(* IEC 61131-3 sources: beebread/doc (part 8) *)

		ELSIF X.STATE = BYTE#2 THEN (* read data *)
			index2 := index + 1; (* PCWORX Workaround *)
			IF X.R_BUF.BUFFER[index] <> ID OR X.R_BUF.BUFFER[index2] <> BYTE#13 THEN (* TYPE DWORD8 *)
				X.ERROR_ID := ID;
			ELSE
				index := index + 2;
				FOR i2 := 1 TO 8 DO;
					ra[i2] := DWORD#0;
					FOR i := 1 TO 4 DO;
						ra[i2] := ra[i2] OR BYTE_TO_DWORD(X.R_BUF.BUFFER[index]);
						ra[i2] := ROR(ra[i2],8);
						index := index + 1;
					END_FOR;
				END_FOR;
				OUT1 := ra[1];
				OUT2 := ra[2];
				OUT3 := ra[3];
				OUT4 := ra[4];
				OUT5 := ra[5];
				OUT6 := ra[6];
				OUT7 := ra[7];
				OUT8 := ra[8];
			END_IF;
		END_IF;
		X.index := index;
	END_IF;
END_IF;
END_FUNCTION_BLOCK

// Commented out for beedance: it uses REAL_TO_DW, which is commented out.
// FUNCTION_BLOCK NET_VAR_REAL8
// VAR_IN_OUT
// 	X : NET_VAR_DATA;
// END_VAR
// VAR_INPUT
// 	IN1 : REAL;
// 	IN2 : REAL;
// 	IN3 : REAL;
// 	IN4 : REAL;
// 	IN5 : REAL;
// 	IN6 : REAL;
// 	IN7 : REAL;
// 	IN8 : REAL;
// END_VAR
// VAR_OUTPUT
// 	OUT1 : REAL;
// 	OUT2 : REAL;
// 	OUT3 : REAL;
// 	OUT4 : REAL;
// 	OUT5 : REAL;
// 	OUT6 : REAL;
// 	OUT7 : REAL;
// 	OUT8 : REAL;
// 	ID : BYTE;
// END_VAR
// VAR
// 	init : BOOL;
// 	i : INT;
// 	i2 : INT;
// 	index : INT;
// 	index2 : INT;
// 	r_dw : DWORD;
// 	ra : ARRAY[1..8] OF REAL;
// END_VAR
//
// IF NOT init THEN
// 	init := TRUE;
// 	X.ID_MAX := X.ID_MAX + USINT#1;
// 	ID := USINT_TO_BYTE(X.ID_MAX);
// END_IF;
//
// IF X.STATE > BYTE#0 AND X.ERROR_ID = BYTE#0 THEN
// 	index := X.index; (* PCWORX Workaround *)
// 	IF INT_TO_UINT(index + 34) > X.BUF_SIZE THEN (* ID (1) + TYPE (1) + 8 x REAL (4) *)
// 		X.ERROR_ID := ID;
// 	ELSE
// 		IF X.STATE = BYTE#1 THEN (* write data *)
// 			ra[1] := IN1;
// 			ra[2] := IN2;
// 			ra[3] := IN3;
// 			ra[4] := IN4;
// 			ra[5] := IN5;
// 			ra[6] := IN6;
// 			ra[7] := IN7;
// 			ra[8] := IN8;
// 			X.S_BUF.BUFFER[index] := ID; (* ID *)
// 			index := index + 1;
// 			X.S_BUF.BUFFER[index] := BYTE#15; (* TYPE REAL8 *)
// 			index := index + 1;
// 			FOR i2 := 1 TO 8 DO;
// 				r_dw := REAL_TO_DW(X:=ra[i2]);
// 				FOR i := 1 TO 4 DO;
// 					X.S_BUF.BUFFER[index] := DWORD_TO_BYTE(r_dw);
// 					r_dw := ROR(r_dw,8);
// 					index := index + 1;
// 				END_FOR;
// 			END_FOR;
//
// 		ELSIF X.STATE = BYTE#2 THEN (* read data *)
// 			index2 := index + 1; (* PCWORX Workaround *)
// 			IF X.R_BUF.BUFFER[index] <> ID OR X.R_BUF.BUFFER[index2] <> BYTE#15 THEN (* TYPE REAL8 *)
// 				X.ERROR_ID := ID;
// 			ELSE
// 				index := index + 2;
// 				FOR i2 := 1 TO 8 DO;
// 					r_dw := DWORD#0;
// 					FOR i := 1 TO 4 DO;
// 						r_dw := r_dw OR BYTE_TO_DWORD(X.R_BUF.BUFFER[index]);
// 						r_dw := ROR(r_dw,8);
// 						index := index + 1;
// 					END_FOR;
// 					ra[i2] := DW_TO_REAL(X:=r_dw);
// 				END_FOR;
// 				OUT1 := ra[1];
// 				OUT2 := ra[2];
// 				OUT3 := ra[3];
// 				OUT4 := ra[4];
// 				OUT5 := ra[5];
// 				OUT6 := ra[6];
// 				OUT7 := ra[7];
// 				OUT8 := ra[8];
// 			END_IF;
// 		END_IF;
// 		X.index := index;
// 	END_IF;
// END_IF;
// END_FUNCTION_BLOCK

// Commented out for beedance: it uses _STRING_TO_BUFFER, which is commented out.
// FUNCTION_BLOCK NET_VAR_STRING
// VAR_IN_OUT
// 	IN : STRING(STRING_LENGTH);
// 	OUT : STRING(STRING_LENGTH);
// 	X : NET_VAR_DATA;
// END_VAR
// VAR_OUTPUT
// 	ID : BYTE;
// END_VAR
// VAR
// 	init : BOOL;
// 	len_str : INT;
// 	index : INT;
// 	index2 : INT;
// END_VAR
//
// IF NOT init THEN
// 	init := TRUE;
// 	X.ID_MAX := X.ID_MAX + USINT#1;
// 	ID := USINT_TO_BYTE(X.ID_MAX);
// END_IF;
//
// IF X.STATE > BYTE#0 AND X.ERROR_ID = BYTE#0 THEN
// 	index := X.index; (* PCWORX Workaround *)
// 	IF X.STATE = BYTE#1 THEN (* write data *)
// 		len_str := LEN(IN);
// 		IF INT_TO_UINT(index + 3 + len_str) > X.BUF_SIZE THEN
// 			X.ERROR_ID := ID;
// 		ELSE
// 			X.S_BUF.BUFFER[index] := ID; (* ID *)
// 			index := index + 1;
// 			X.S_BUF.BUFFER[index] := BYTE#6; (* TYPE REAL *)
// 			index := index + 1;
// 			X.S_BUF.BUFFER[index] := INT_TO_BYTE(len_str); (* number of bytes *)
// 			index := index + 1;
// 			_STRING_TO_BUFFER(STR:=IN,POS:=index,PT:=REF(X.S_BUF.BUFFER),SIZE:=X.BUF_SIZE);
// 			index := index + len_str;
// 		END_IF;
// 	ELSIF X.STATE = BYTE#2 THEN (* read data *)
// 		index2 := index + 1; (* PCWORX Workaround *)
// 		IF X.R_BUF.BUFFER[index] <> ID OR X.R_BUF.BUFFER[index2] <> BYTE#6 THEN
// 			X.ERROR_ID := ID;
// 		ELSE
// 			index := index + 2;
// 			len_str := BYTE_TO_INT(X.R_BUF.BUFFER[index]);
// 			index2 := index + 1;
// 			index := index2 + len_str;
// 			IF len_STR > 0 THEN
// 				OUT := BUFFER_TO_STRING(PT:=REF(X.R_BUF.BUFFER),SIZE:=X.BUF_SIZE,START:=INT_TO_UINT(index2),STOP:=INT_TO_UINT(index - 1));
// 			ELSE
// 				OUT := '';
// 			END_IF;
// 		END_IF;
// 	END_IF;
// 	X.index := index;
// END_IF;
// END_FUNCTION_BLOCK

// Commented out for beedance: it uses REAL_TO_DW, which is commented out.
// FUNCTION_BLOCK NET_VAR_X8
// VAR_IN_OUT
// 	X : NET_VAR_DATA;
// END_VAR
// VAR_INPUT
// 	IN_REAL1 : REAL;
// 	IN_REAL2 : REAL;
// 	IN_DINT1 : DINT;
// 	IN_DINT2 : DINT;
// 	IN_UDINT1 : UDINT;
// 	IN_UDINT2 : UDINT;
// 	IN_DWORD1 : DWORD;
// 	IN_DWORD2 : DWORD;
// END_VAR
// VAR_OUTPUT
// 	OUT_REAL1 : REAL;
// 	OUT_REAL2: REAL;
// 	OUT_DINT1 : DINT;
// 	OUT_DINT2 : DINT;
// 	OUT_UDINT1 : UDINT;
// 	OUT_UDINT2 : UDINT;
// 	OUT_DWORD1 : DWORD;
// 	OUT_DWORD2 : DWORD;
// 	ID : BYTE;
// END_VAR
// VAR
// 	init : BOOL;
// 	i : INT;
// 	i2 : INT;
// 	index : INT;
// 	index2 : INT;
// 	ra : ARRAY[1..8] OF DWORD;
// END_VAR
//
// IF NOT init THEN
// 	init := TRUE;
// 	X.ID_MAX := X.ID_MAX + USINT#1;
// 	ID := USINT_TO_BYTE(X.ID_MAX);
// END_IF;
//
// IF X.STATE > BYTE#0 AND X.ERROR_ID = BYTE#0 THEN
// 	index := X.index; (* PCWORX Workaround *)
// 	IF INT_TO_UINT(index + 34) > X.BUF_SIZE THEN  (* ID (1) + TYPE (1) + 8 x DWORD (4) *)
// 		X.ERROR_ID := ID;
// 	ELSE
// 		IF X.STATE = BYTE#1 THEN (* write data *)
// 			ra[1] := REAL_TO_DW(X:=IN_REAL1);
// 			ra[2] := REAL_TO_DW(X:=IN_REAL2);
// 			ra[3] := DINT_TO_DWORD(IN_DINT1);
// 			ra[4] := DINT_TO_DWORD(IN_DINT2);
// 			ra[5] := UDINT_TO_DWORD(IN_UDINT1);
// 			ra[6] := UDINT_TO_DWORD(IN_UDINT2);
// 			ra[7] := IN_DWORD1;
// 			ra[8] := IN_DWORD2;
// 			X.S_BUF.BUFFER[index] := ID; (* ID *)
// 			index := index + 1;
// 			X.S_BUF.BUFFER[index] := BYTE#21; (* TYPE X8 *)
// 			index := index + 1;
// 			FOR i2 := 1 TO 8 DO;
// 				FOR i := 1 TO 4 DO;
// 					X.S_BUF.BUFFER[index] := DWORD_TO_BYTE(ra[i2]);
// 					ra[i2] := ROR(ra[i2],8);
// 					index := index + 1;
// 				END_FOR;
// 			END_FOR;
//
// 		ELSIF X.STATE = BYTE#2 THEN (* read data *)
// 			index2 := index + 1; (* PCWORX Workaround *)
// 			IF X.R_BUF.BUFFER[index] <> ID OR X.R_BUF.BUFFER[index2] <> BYTE#21 THEN (* TYPE X8 *)
// 				X.ERROR_ID := ID;
// 			ELSE
// 				index := index + 2;
// 				FOR i2 := 1 TO 8 DO;
// 					ra[i2] := DWORD#0;
// 					FOR i := 1 TO 4 DO;
// 						ra[i2] := ra[i2] OR BYTE_TO_DWORD(X.R_BUF.BUFFER[index]);
// 						ra[i2] := ROR(ra[i2],8);
// 						index := index + 1;
// 					END_FOR;
// 				END_FOR;
// 				OUT_REAL1 := DW_TO_REAL(X:=ra[1]);
// 				OUT_REAL2 := DW_TO_REAL(X:=ra[2]);
// 				OUT_DINT1 := DWORD_TO_DINT(ra[3]);
// 				OUT_DINT2 := DWORD_TO_DINT(ra[4]);
// 				OUT_UDINT1 := DWORD_TO_UDINT(ra[5]);
// 				OUT_UDINT2 := DWORD_TO_UDINT(ra[6]);
// 				OUT_DWORD1 := ra[7];
// 				OUT_DWORD2 := ra[8];
// 			END_IF;
// 		END_IF;
// 		X.index := index;
// 	END_IF;
// END_IF;
// END_FUNCTION_BLOCK

FUNCTION NETWORK_VERSION : DWORD
VAR_INPUT
	IN : BOOL;
END_VAR

IF in THEN
	NETWORK_VERSION := DATE_TO_DWORD(D#2016-07-01);
ELSE
	NETWORK_VERSION := 135;
END_IF;
END_FUNCTION

// Commented out for beedance: it uses CODE, which is commented out.
// FUNCTION_BLOCK PRINT_SF
// VAR_IN_OUT
// 	PRINTF_DATA : PRINTF_DATA;
// 	STR : STRING(LOG_SIZE);
// END_VAR
// VAR
// 	pos : INT;
// 	c : INT;
// 	src : STRING(1) := '~';
// 	run : BOOL;
// END_VAR
//
// IF LEN(STR) > 0 THEN
// 	run := TRUE;
//
// 	WHILE (run) DO
// 		pos := FIND(STR,src);
// 		PRINTF_DATA[10] := '';
//
// 		IF pos = 0 THEN
// 			run:= FALSE;
// 		ELSE
// 			c := CODE(STR:=STR,POS:=pos + 1);
// 			IF ISC_NUM(INT_TO_BYTE(c)) THEN
// 				c := c - 48; (* necessary because only one var is allowed inside an index expression *)
// 				PRINTF_DATA[10] := PRINTF_DATA[c]; (* command 1-9 gives parameter index 1-9 *)
// 				(* replace parameter with text *)
// 			END_IF;
// 			IF LEN(PRINTF_DATA[10]) + LEN(STR) > LOG_SIZE THEN
// 				PRINTF_DATA[10] := '..';
// 			END_IF;
// 			(* pcworx: output and input string must be different *)
// 			PRINTF_DATA[11] := STR;
// 			STR := REPLACE(PRINTF_DATA[11],PRINTF_DATA[10],2,pos);
// 		END_IF;
// 	END_WHILE;
// END_IF;
// END_FUNCTION_BLOCK

// Commented out for beedance: it uses CODE, which is commented out.
// FUNCTION_BLOCK RC4_CRYPT_STREAM
// VAR_IN_OUT
// 	MODE : INT;
// 	KEY : STRING(40);
// 	BUF : ARRAY [0..63] OF BYTE;
// 	SIZE : UDINT;
// END_VAR
//
// VAR_OUTPUT
// 	POS : UDINT;
// END_VAR
//
// VAR
// 	sbox : ARRAY [0..255] OF BYTE;
// 	skey : ARRAY [0..255] OF BYTE;
// 	a : INT;
// 	b : INT;
// 	c : INT;
// 	d : USINT;
// 	e : USINT;
// 	end : UDINT;
// 	v : BYTE;
// END_VAR
//
// CASE MODE OF
//
// 1:	(* initialization *)
// 	b := LEN(KEY) - 1;
// 	IF b < 0 OR SIZE < 1 THEN
// 		MODE := 3;
// 		RETURN;
// 	END_IF;
//
// 	FOR a := 0 TO b DO
// 		skey[a] := CODE(KEY, a + 1);
// 		sbox[a] := INT_TO_BYTE(a);
// 	END_FOR;
//
// 	c := 0;
// 	FOR a := b + 1 TO 255 DO
// 		skey[a] := skey[c];
// 		sbox[a] := INT_TO_BYTE(a);
// 		c := c + 1;
// 		IF c > b THEN c := 0; END_IF;
// 	END_FOR;
//
// 	d := 0;
// 	FOR a := 0 TO 255 DO
// 		d := d + sbox[a] + skey[a];
// 		v := sbox[a];
// 		sbox[a] := sbox[d];
// 		sbox[d] := v;
// 	END_FOR;
//
// 	POS := 0;
// 	end := SIZE;
// 	SIZE := MIN(64,end);
// 	d := 0;
// 	e := 0;
// 	MODE := 2;
//
// 2:	(* encrypt/decrypt data *)
//
// 	b := UDINT_TO_INT(SIZE) - 1;
// 	FOR a := 0 TO b DO
// 		d := d + 1;
// 		e := e + sbox[d];
// 		v := sbox[d];
// 		sbox[d] := sbox[e];
// 		sbox[e] := v;
// 		v := sbox[d] + sbox[e];
// 		BUF[a] :=BUF[a] XOR sbox[v];
// 	END_FOR;
//
// 	POS := POS + SIZE;
// 	SIZE := MIN(64,end - POS);
//
// 	IF SIZE = 0 THEN
// 		MODE := 3;
// 	END_IF;
// END_CASE;
// END_FUNCTION_BLOCK

// Commented out for beedance: it uses BUFFER_SEARCH, which is commented out.
// FUNCTION_BLOCK READ_HTTP
// VAR_INPUT
// 	SIZE : UINT;
// 	POS : INT;
// 	SRC : STRING;
// END_VAR
// VAR_IN_OUT
// 	PT : NW_BUF_LONG;
// END_VAR
// VAR_OUTPUT
// 	READ_HTTP : STRING(STRING_LENGTH);
// END_VAR
// VAR
// 	index : INT;
// 	s1 : INT;
// 	e1 : INT;
// 	stop : INT;
// END_VAR
//
// stop := UINT_TO_INT(SIZE) - 1;
//
// IF LEN(SRC) = 0 THEN
// 	(* if there is no search term, evaluate the HTTP STATUS *)
// 	SRC := 'HTTP/'; (* new search term *)
// ELSE
// 	(* append the searched parameter text *)
// 	SRC := CONCAT(SRC,': ');
// END_IF;
//
// s1 := BUFFER_SEARCH(pt:=REF(PT),SIZE:=SIZE,STR:=SRC,POS:=POS,IGN:=TRUE);
//
// IF s1 >= 0 THEN (* Text found *)
// 	e1 := s1;
//
// 	(* search start of line *)
// 	index := s1 - 1;
// 	WHILE (index > 0) DO
// 		IF pt[index] < BYTE#32 THEN EXIT; END_IF;
// 		s1 := s1 - 1;
// 		index := index - 1;
// 	END_WHILE;
//
// 	(* search end of line *)
// 	index := e1 + 1;
// 	WHILE (index <= stop) DO
// 		IF pt[index] < BYTE#32 THEN EXIT; END_IF;
// 		e1 := e1 + 1;
// 		index := index + 1;
// 	END_WHILE;
//
// 	s1 := s1 + LEN(SRC); (* do not copy 'search term: ' *)
//
// 	(* copy string *)
// 	READ_HTTP := BUFFER_TO_STRING(PT:=REF(PT),SIZE:=SIZE,START:=s1,STOP:=e1);
// ELSE
// 	READ_HTTP := '';
// END_IF;
// END_FUNCTION_BLOCK

// Commented out for beedance: it uses _STRING_TO_BUFFER, which is commented out.
// FUNCTION_BLOCK SHA1_STR
// VAR_INPUT
// 	RUN: BOOL;
// END_VAR
// VAR_OUTPUT
// 	DONE: BOOL;
// END_VAR
// VAR_IN_OUT
// 	STR: STRING(STRING_LENGTH);
// 	SHA1 : ARRAY [0..19] OF BYTE;
// END_VAR
//
// VAR
// 	run_last: BOOL;
// 	SHA1_STREAM : SHA1_STREAM;
// 	buf : ARRAY [0..63] OF BYTE;
// 	mode : INT;
// 	size : UDINT;
// 	pos : UDINT;
// END_VAR
//
// CASE mode OF
// 0:	(* wait for start *)
// 	IF RUN AND NOT run_last THEN
// 		DONE := FALSE;
// 		mode := 1; (* initialization *)
// 		size := LEN(STR);
// 	END_IF;
//
// 2:	(* Data copy and Calc *)
// 	IF size > 0 THEN
// 		_STRING_TO_BUFFER(STR:=MID(STR, UDINT_TO_INT(SIZE), UDINT_TO_INT(POS) + 1), POS:=0, PT:=REF(buf), SIZE:=SIZEOF(buf));
// 	END_IF;
//
// 3:	DONE := TRUE;
// 	mode := 0; (* Stop *)
//
// END_CASE;
//
// IF mode > 0 THEN
// 	SHA1_STREAM(SIZE:=size, MODE:=mode, BUF:=buf, SHA1:=SHA1, POS=>pos);
// END_IF;
//
// run_last := RUN;
// END_FUNCTION_BLOCK

FUNCTION_BLOCK SHA1_STREAM
VAR_IN_OUT
	MODE : INT;
	BUF : ARRAY [0..63] OF BYTE;
	SHA1 : ARRAY [0..19] OF BYTE;
	SIZE : UDINT;
END_VAR

VAR_OUTPUT
	POS : UDINT;
END_VAR

VAR
	hash : ARRAY [0..4] OF DWORD;
	end : UDINT;
	block : UDINT;
	pad_1 : BOOL;
	w : ARRAY [0..79] OF DWORD;
	n : INT;
	n1 : INT;
	a : DWORD;
	b : DWORD;
	c : DWORD;
	d : DWORD;
	e : DWORD;
	f : DWORD;
	k : DWORD;
	x : DWORD;
	z : INT;
END_VAR

CASE MODE OF

1:	(* initialization of the hash values *)
	hash[0] := DWORD#16#67452301;
	hash[1] := DWORD#16#EFCDAB89;
	hash[2] := DWORD#16#98BADCFE;
	hash[3] := DWORD#16#10325476;
	hash[4] := DWORD#16#C3D2E1F0;

	(* initialize buffer *)
	FOR n := 16 TO 79 DO
   		w[n] := DWORD#0;
	END_FOR;

	block := SHR(SIZE,6) + BOOL_TO_UDINT((UDINT_TO_BYTE(SIZE) AND 16#3F) > 55);	(* calculate the required blocks *)

	pad_1 := FALSE;
	POS := 0;
	End := SIZE;
	SIZE := MIN(64,End);
	MODE := 2;

2:	FOR n := UDINT_TO_INT(SIZE) TO 63 DO (* append padding bytes *)
		BUF[n] := 0;
	END_FOR;

	IF SIZE < 64 AND NOT pad_1 THEN
		BUF[SIZE] := 2#1000_0000;
		pad_1 := TRUE;
	END_IF;

	POS := POS + SIZE;
	SIZE := MIN(64,End - POS);

	n := 0;	(* copy byte array into DWORD array *)
	FOR n1 := 0 TO 15 DO
		w[n1] := DWORD_OF_BYTE(BUF[n],BUF[n+1],BUF[n+2],BUF[n+3]);
		n := n + 4;
	END_FOR;

	IF block = 0 THEN (* enter the data length at the end of the last block *)
		w[15] := SHL(UDINT_TO_DWORD(End),3); (* enter the number of data bits *)
		MODE := 3;
	ELSE
		block := block - 1;
	END_IF;

	FOR n := 16 TO 79 DO (* extend the 16 32-bit words to 80 32-bit words *)
		w[n] := ROL(w[n-3] XOR w[n-8] XOR w[n-14] XOR w[n-16],1);
	END_FOR;

	a := hash[0];
	b := hash[1];
	c := hash[2];
	d := hash[3];
	e := hash[4];

	FOR n := 0 TO 79 DO
		IF n <= 19 THEN
			f := (b AND c) OR (NOT(b) AND d);
			k := DWORD#16#5A827999;
		ELSIF n <= 39 THEN
			f := b XOR c XOR d;
			k := DWORD#16#6ED9EBA1;
		ELSIF n <= 59 THEN
			f := (b AND c) OR (b AND d) OR (c AND d);
			k := DWORD#16#8F1BBCDC;
		ELSE
			f := b XOR c XOR d;
			k := DWORD#16#CA62C1D6;
		END_IF;

		x := ROL(a,5) + f + e + k + w[n];
		e := d;
		d := c;
		c := ROL(b,30);
		b := a;
		a := x;
	END_FOR;

	(* add the current hash values to the last value *)
	hash[0] := hash[0] + a;
	hash[1] := hash[1] + b;
	hash[2] := hash[2] + c;
	hash[3] := hash[3] + d;
	hash[4] := hash[4] + e;

END_CASE;

IF MODE = 3 THEN
	z := 0;
	FOR n := 0 TO 4 DO (* convert DWORD to BYTE array *)
		FOR n1 := 0 TO 3 DO
			hash[n] := ROL(hash[n],8);
			SHA1[z] := DWORD_TO_BYTE(hash[n]);
			z := z + 1;
		END_FOR;
	END_FOR;
END_IF;
END_FUNCTION_BLOCK

// Commented out for beedance: it computes with pointers as addresses (pt := pt + 1); beedance references (REF_TO) have no arithmetic.
// FUNCTION SHA1_TO_STRH : STRING(40)
// VAR_INPUT
// 	SHA1 : ARRAY [0..19] OF BYTE;
// END_VAR
// VAR
// 	i : INT;
// 	tmp : BYTE;
// 	pt : REF_TO BYTE;
// END_VAR
// pt := REF(SHA1_TO_STRH); (* read output adress to pointer *)
//
// FOR i := 0 TO 19 DO; (* write the 10 hex characters backwards *)
// 	tmp := SHR(SHA1[i],4);
// 	PT^ := tmp + SEL(tmp <= 9,87,48);
// 	pt := pt + 1; (* decrement the pointer *)
// 	tmp := SHA1[i] AND 2#1111;
// 	PT^ := tmp + SEL(tmp <= 9,87,48);
// 	pt := pt + 1; (* decrement the pointer *)
// END_FOR;
// pt^:= 0; (* write the closing byte for the string *)
// END_FUNCTION

// Commented out for beedance: it has a comment between UNTIL and END_REPEAT, which beedance does not parse yet.
// FUNCTION_BLOCK SMTP_CLIENT
// VAR_INPUT
// 	ACTIVATE : BOOL;
// 	TIMEOUT : TIME;
// 	DTI : DT;
// 	DTI_OFFSET : INT;
// 	DNS_IP4 : DWORD;
// END_VAR
// VAR_OUTPUT
// 	DONE : BOOL;
// 	BUSY : BOOL;
// 	ERROR_C : DWORD;
// 	ERROR_T : BYTE;
// END_VAR
// VAR_IN_OUT
// 	SERVER : STRING;
// 	MAILFROM : STRING;
// 	MAILTO : STRING(STRING_LENGTH);
// 	SUBJECT : STRING;
// 	BODY : STRING(STRING_LENGTH);
// 	FILES : STRING(STRING_LENGTH);
// END_VAR
// VAR
// 	IP_C : IP_C; (* IP_Control management structure *)
// 	S_BUF : NETWORK_BUFFER;
// 	R_BUF : NETWORK_BUFFER;
// 	F_BUF : NETWORK_BUFFER;
// 	URL_DATA : url;
// 	DNS_CLIENT : DNS_CLIENT;
// 	IPC : IP_CONTROL;
// 	FS : FILE_SERVER;
// 	FSD : FILE_SERVER_DATA;
// 	BASE64_ENCODE_STR : BASE64_ENCODE_STR;
// 	BASE64_ENCODE_STREAM : BASE64_ENCODE_STREAM;
// 	fpd : FILE_PATH_DATA;
// 	MD5_CRAM_AUTH : MD5_CRAM_AUTH;
// 	MD5_RUN : BOOL;
// 	activate_last : BOOL;
// 	step : INT;
// 	snd_step : INT;
// 	str1 : STRING(STRING_LENGTH);
// 	str2 : STRING(STRING_LENGTH);
// 	str3 : STRING;
// 	snd_text :	STRING(STRING_LENGTH);
// 	snd_lf_cnt : INT;
// 	rcv_text :	STRING(STRING_LENGTH);
// 	rcv_s : STRING(3);
// 	rcv_state : INT;
// 	auth_names : STRING := ' PLAIN; LOGIN; CRAM-MD5';
// 	auth_names_tls : STRING := ' PLAIN; LOGIN; CRAM-MD5;STARTTLS';
// 	auth_state : BYTE;
// 	TON_WAIT : TON;
// 	last_step : INT;
// 	next_step : INT;
// 	timeout2 : TIME;
// 	timeout3 : TIME;
// 	last_block : BOOL;
// 	file_delete : BOOL;
// 	esmtp : BOOL;
// 	cnt1 : INT;
// 	cnt2 : INT;
// 	cnt3 : INT;
// 	cnt4 : INT;
// 	idx1 : INT;
// 	idx2 : INT;
// 	idx3 : INT;
// 	snd_idx : INT;
// 	snd_enable : BOOL;
// 	i1 : INT;
// 	b64_done : BOOL;
// 	b64_start : BOOL;
// 	b64_max : UINT := 2880; (* short = 960 / long = 2880 *)
// 	b64_buf1 : ARRAY [0..47] OF BYTE;
// 	b64_buf2 : ARRAY [0..63] OF BYTE;
// 	b64_size1 : INT;
// 	b64_size2 : INT;
// 	b64_lf : BOOL;
// 	b64_str1	: STRING(144);
// 	b64_str2	: STRING(192);
// 	md5_user : STRING(64);
// 	md5_password : STRING(64);
// 	md5_b64_ts : STRING(64);
// 	md5_auth_key : STRING(192);
// 	ip_c_red_disable : BOOL; (* IP_CONTROL - suppress remote disconnect error *)
// 	ssl_mode :	BYTE;(*SSL/TLS Mode -   0 = off / 1 = SSL / 2 = TLS*)
//
// 	(*LOG_MSG : LOG_MSG;
// 	_debug_enable : BOOL := TRUE;*)
// END_VAR
//
// CASE step OF
//
// 00:
// 	IF ACTIVATE AND NOT activate_last THEN
// 		TIMEOUT := MAX(T#10s,TIMEOUT);
// 		timeout2 := TIMEOUT + T#1s;
// 		timeout3 := TIMEOUT / 2;
// 		DONE := FALSE;
// 		ip_c_red_disable := FALSE;
// 		ERROR_C := DWORD#0;
// 		ERROR_T := BYTE#0;
// 		FSD.ERROR := BYTE#0;
// 		file_delete := FALSE;
// 		URL_DATA := STRING_TO_URL(STR:=SERVER,DEFAULT_PROTOCOL:='',DEFAULT_PATH:='/');
// 		idx1 := FIND(URL_DATA.USER,'%'); (* change % character to @ *)
// 		IF idx1 > 0 THEN
// 			URL_DATA.USER := REPLACE(URL_DATA.USER,'@',1,idx1);
// 		END_IF;
// 		esmtp := LEN(URL_DATA.PASSWORD) > 0; (* SMTP or ExtendedSMTP *)
// 		step := 10;
// 	END_IF;
//
// 10:
// 	IF DNS_CLIENT.DONE THEN
// 		step := 20;
// 	ELSIF DNS_CLIENT.ERROR <> DWORD#0 THEN
// 		ERROR_C := DNS_CLIENT.ERROR;
// 		ERROR_T := BYTE#1;
// 		step := 980;
// 	END_IF;
//
// 20:	(* set up SMTP communication *)
// 	IF FIND(';SSL;ssl;Ssl', URL_DATA.PROTOCOL) > 1 THEN
// 		ssl_mode := BYTE#1;
// 		IP_C.C_PORT := SEL(URL_DATA.PORT = WORD#0,URL_DATA.PORT,WORD#465); (* enter port number *)
// 		IP_C.MAILBOX[16] := BYTE#1; (* enable SSL mode *)
// 	ELSIF FIND(';TLS;tls;Tls', URL_DATA.PROTOCOL) > 1 THEN
// 		ssl_mode := BYTE#2;
// 		IP_C.C_PORT := SEL(URL_DATA.PORT = WORD#0,URL_DATA.PORT,WORD#587); (* enter port number *)
// 		IP_C.MAILBOX[16] := BYTE#0; (* no SSL mode yet*)
// 	ELSE
// 		ssl_mode := BYTE#0;
// 		IP_C.C_PORT := SEL(URL_DATA.PORT = WORD#0,URL_DATA.PORT,WORD#25); (* enter port number *)
// 		IP_C.MAILBOX[16] := BYTE#0; (* no SSL mode*)
// 	END_IF;
//
//   	IP_C.C_IP := DNS_CLIENT.IP4; (* enter IP *)
//   	IP_C.C_MODE := BYTE#0; (* Mode: TCP+ACTIV+PORT *)
//   	IP_C.TIME_RESET := TRUE; (* reset timeout monitoring *)
//   	IP_C.C_ENABLE := TRUE; (* enable connection setup *)
//   	IP_C.R_OBSERVE := TRUE; (* receive monitoring *)
// 	IP_C.MAILBOX[3] := BYTE#0; (* re-enable IP receive *)
// 	R_BUF.SIZE := UINT#0;
// 	snd_enable := TRUE; (* allow immediate sending *)
// 	snd_idx := 0;
// 	step := 30;
//
// 30:
// 	IF rcv_state = 220 THEN (* 220 = Service ready *)
// 		IF esmtp THEN
// 			snd_text := 'EHLO OSCAT'; (* ExtendedSMTP *)
//
// 			str1:= SEL(ssl_mode = BYTE#2,auth_names,auth_names_tls);
// 			auth_state := BYTE#0;
// 			idx2 := 1900;
//
// 			next_step := 40;
// 		ELSE
// 			snd_text := 'HELO OSCAT'; (* SMTP *)
// 			next_step := 90;
// 		END_IF;
// 		snd_lf_cnt := 1;
// 	END_IF;
//
// 40:
// 	IF rcv_state = 250 THEN
// 		(* 250 = Requested mail action okay, complete
// 			1. some providers do not announce an AUTH method with SSL.
// 			2. since some SMTP servers send the 250 xxx messages in more than one telegram,
// 		       a special SSL handling must be done via timeout monitoring instead *)
// 		IF ssl_mode >= BYTE#1 AND TON_WAIT.ET > T#1s THEN
// 			rcv_text := '250-AUTH LOGIN'; (* fake AUTH *)
//
//         	(*####################  DEBUG-MESSAGE  ###################################*)
// 			(*IF _debug_enable THEN
// 				LOG_CL.NEW_MSG := 'SMTP: PROBLEM /rcv_text ~1';
// 				LOG_CL.PRINTF[1] := rcv_text;
// 				LOG_MSG();
// 			END_IF;*)
// 			(*########################################################################*)
//
// 		END_IF;
//
// 		IF FIND(rcv_text,'AUTH') > 0 THEN (* BUGFIX  !*)
// 			IP_C.MAILBOX[3] := BYTE#1; (* block IP receive until data has been checked *)
// 			idx1 := 0;
// 			step := 50;
// 		END_IF;
//
// 	END_IF;
//
// 50:
// 	str2 := ELEMENT_GET(59, idx1, str1); (* separator >;< *)
//
// 	(*####################  DEBUG-MESSAGE  ###################################*)
// 	(*IF _debug_enable THEN
// 		LOG_CL.NEW_MSG := 'ST s1>~1< s2>~2< i1>~2< ~3';
// 		LOG_CL.PRINTF[1] := str1;
// 		LOG_CL.PRINTF[2] := str2;
// 		LOG_CL.PRINTF[3] := INT_TO_STRING(idx1);
// 		LOG_CL.PRINTF[4] := rcv_text;
// 		LOG_MSG();
// 	END_IF;*)
// 	(*########################################################################*)
//
// 	IF LEN(str2) > 0 THEN
// 		IF FIND(rcv_text,str2) > 0 THEN
// 			auth_state := BIT_LOAD_B(auth_state, TRUE, idx1);
// 			str3 := str2; (* save current AUTH type name *)
// 			idx2 := 1000 + (idx1 * 100); (* calculate step *)
// 		END_IF;
// 		idx1 := idx1 + 1;
// 	ELSE
// 		IF auth_state <> BYTE#0 THEN (* AUTH type found *)
// 			IP_C.MAILBOX[3] := BYTE#0; (* re-enable IP receive *)
// 			(* mit den jeweiligen Authentifizierung Schritten fortfahren:
// 			   1000 = PLAIN / 1100 = LOGIN / 1200 = CRAM-MD5 / 1300 TLS *)
// 			step := idx2;
// 		ELSE
// 			idx1 := 0;
// 			rcv_text := '';
// 			IP_C.MAILBOX[3] := BYTE#0; (* re-enable IP receive *)
// 			step := 40; (* wait for the next 250 auth message *)
// 		END_IF;
// 	END_IF;
//
// 	(*####################  DEBUG-MESSAGE  ###################################*)
// 	(*IF _debug_enable THEN
// 		LOG_CL.NEW_MSG := 'SMTP: /auth ~1 /idx1 ~2 /idx2 ~3 /str3 ~4 /LEN ~5 /step ~6 /str1 ~7';
// 		LOG_CL.PRINTF[1] := BYTE_TO_STRING(auth_state);
// 		LOG_CL.PRINTF[2] := INT_TO_STRING(idx1);
// 		LOG_CL.PRINTF[3] := INT_TO_STRING(idx2);
// 		LOG_CL.PRINTF[4] := str3;
// 		LOG_CL.PRINTF[5] := INT_TO_STRING(LEN(str2));
// 		LOG_CL.PRINTF[6] := INT_TO_STRING(step);
// 		LOG_CL.PRINTF[7] := str1;
// 		LOG_MSG();
// 	END_IF;*)
// 	(*########################################################################*)
//
//  (* ++++++++++++++++++++++++++++++++++++++++++++++++++++++*)
//
// 90:
// 	IF rcv_state = 235 OR rcv_state = 250 THEN (* 235 = Authentication successful / 250 Requested mail action okay *)
// 		str2 := MAILFROM;
// 		str1 := ELEMENT_GET(59, 0, str2);(* read MAILFROM, separator >;< *)
// 		snd_text := INSERT('MAIL FROM: <>', str1, 12);
// 		str3 := REPLACE(snd_text, 'From', 9, 1); (* replace 'MAIL FROM' with "From" and buffer it *)
// 		next_step := 95;
// 		cnt1 := ELEMENT_COUNT(35, MAILTO); (* separator >#<, determine the number of blocks *)
// 		cnt2 := 0;
// 	END_IF;
//
// 95:
// 	IF rcv_state = 250 THEN (* 250 = Requested mail action okay *)
// 		IF cnt2 < cnt1 THEN
// 			str1 := ELEMENT_GET(35, cnt2, MAILTO);(* separator >#< *)
// 			cnt3 := ELEMENT_COUNT(59, str1); (* separator >;<, determine the number of sub-blocks *)
// 			cnt4 := 0;
// 			cnt2 := cnt2 + 1;
// 			step := 100; (* evaluate block content *)
// 		ELSE
// 			step := 110; (* all blocks processed *)
// 		END_IF;
// 	END_IF;
//
// 100:
// 	IF rcv_state = 250 THEN (* 250 = Requested mail action okay *)
// 		IF cnt4 < cnt3 THEN
// 			str2 := ELEMENT_GET(59, cnt4, str1); (* separator >;< *)
// 			snd_text := INSERT('RCPT TO: <>', str2, 10);
// 			cnt4 := cnt4 + 1;
// 			next_step := 100;
// 		ELSE
// 			step := 95;
// 		END_IF;
// 	END_IF;
//
// 110:
// 	IF rcv_state = 250 THEN (* 250 = Requested mail action okay *)
// 		snd_text := 'DATA';
// 		next_step := 120;
// 	END_IF;
//
// 120:
// 	IF rcv_state = 354 THEN (* 354 = Start mail input; end with. *)
// 		snd_enable := FALSE;
// 		str2 := MAILFROM;
// 		str1 := ELEMENT_GET(59, 1, str2);(* read display name, separator >;< *)
// 		IF LEN(str1) > 0 THEN
// 			str2 := INSERT('"" ', str1, 1);
// 			snd_text := INSERT(str3, str2, 6);
// 		ELSE
// 			snd_text := str3;
// 		END_IF;
// 		cnt2 := 0;
// 		cnt1 := MIN(2,cnt1); (* hide blind copy block *)
// 		step := 200;
// 	END_IF;
//
// 200:
// 	IF snd_step = 0 THEN
// 		IF cnt2 < cnt1 THEN
// 			str1 := ELEMENT_GET(35, cnt2, MAILTO);(* separator >#< *)
// 			cnt3 := ELEMENT_COUNT(59, str1); (* separator >;<, determine the number of sub-blocks *)
// 			cnt4 := 0;
// 			cnt2 := cnt2 + 1;
// 			str3 := SEL(cnt2 = 1,'Cc: <>','To: <>');
// 			step := 205; (* evaluate block content *)
// 		ELSE
// 			step := 210; (* all blocks processed *)
// 		END_IF;
// 	END_IF;
//
// 205:
// 	IF snd_step = 0 THEN
// 		IF cnt4 < cnt3 THEN
// 			str2 := ELEMENT_GET(59, cnt4, str1); (* separator >;< *)
// 			snd_text := INSERT(str3, str2, 5);
// 			cnt4 := cnt4 + 1;
// 		ELSE
// 			step := 200;
// 		END_IF;
// 	END_IF;
//
// 210:
// 	IF snd_step = 0 THEN
// 		snd_text := CONCAT('Subject: ',SUBJECT);
// 		step := 220;
// 	END_IF;
//
// 220:
// 	IF snd_step = 0 THEN
// 		DTI := UDINT_TO_DT(DT_TO_UDINT(DTI) + INT_TO_UDINT(- DTI_OFFSET * 60)); (* convert minute offset to seconds and add *)
// 		IF esmtp THEN (* ESMTP Format >Date: Thu, 21 May 1998 05:33:29 -0700< *)
// 			str2 := ';Mon;Tue;Wed;Thu;Fri;Sat;Sun';
// 			str1 := ELEMENT_GET(59, DAY_OF_WEEK(DT_TO_DATE(DTI)), str2);
// 			snd_text := CONCAT('Date: ',str1);
// 			str1 := DT_TO_STRF(DTI, 0, ', #H #E #A #N:#R:#T +0000', 1);
// 			snd_text := CONCAT(snd_text,str1);
// 		ELSE (* SMTP Format >Date: 21 May 98 05:33:29< *)
// 			snd_text := DT_TO_STRF(DTI, 0, 'Date: #G #E #B #N:#R:#T', 1);
// 		END_IF;
// 		step := 230;
// 	END_IF;
//
// 230:
// 	IF snd_step = 0 THEN
// 		snd_text := 'MIME-Version: 1.0';
// 		step := 250;
// 	END_IF;
//
// 250:
// 	IF snd_step = 0 THEN
// 		snd_text := 'Content-Type: multipart/mixed;boundary="x"';
// 		snd_lf_cnt := 2;
// 		step := 260;
// 	END_IF;
//
// 260:
// 	IF snd_step = 0 THEN
// 		snd_enable := TRUE;
// 		snd_text := 'This is a multi-part message in MIME format.';
// 		step := 270;
// 	END_IF;
//
// 270:
// 	IF snd_step = 0 THEN
// 		snd_enable := FALSE;
// 		snd_text := '--x';
// 		snd_lf_cnt := 1;
// 		step := 280;
// 	END_IF;
//
// 280:
// 	IF snd_step = 0 THEN
// 		snd_text := 'Content-Type: text/plain; format=flowed; charset="iso-8859-1";';
// 		snd_text := CONCAT(snd_text,' reply-type=original'); (* PCWORX only supports constants with max 80 characters *)
// 		step := 290;
// 	END_IF;
//
// 290:
// 	IF snd_step = 0 THEN
// 		snd_text := 'Content-Transfer-Encoding: 8bit';
// 		snd_lf_cnt := 2;
// 		step := 300;
// 	END_IF;
//
// 300:
// 	IF snd_step = 0 THEN
// 		snd_enable := TRUE;
// 		snd_text := BODY;
// 		snd_lf_cnt := 2;
// 		step := 310;
// 	END_IF;
//
// 310:
// 	IF snd_step = 0 THEN
// 		cnt1 := ELEMENT_COUNT(59, FILES) - 1; (* number of files *)
// 		step := 400;
// 	END_IF;
//
// (* +++++++++++++ File-Attachment ++++++++++++ *)
// 400:
// 	IF cnt1 >= 0 THEN
// 		str1 := ELEMENT_GET(59, cnt1, FILES);
// 		FILE_PATH_SPLIT(FILENAME:=str1,X:=fpd); (* split file path *)
// 		IF fpd.FILENAME = '#DEL#' THEN
// 			file_delete := TRUE;
// 		ELSE
// 			step := 410;
// 		END_IF;
// 		cnt1 := cnt1 - 1;
// 	ELSE
// 		step := 800;
// 	END_IF;
//
// 410:
// 	IF snd_step = 0 THEN
// 		snd_enable := FALSE;
// 		snd_text := '--x';
// 		snd_lf_cnt := 1;
// 		step := 420;
// 	END_IF;
//
// 420:
// 	IF snd_step = 0 THEN
// 		snd_text := 'Content-Transfer-Encoding: BASE64';
// 		str2 := CONCAT(fpd.FILENAME,'"');
// 		step := 430;
// 	END_IF;
//
// 430:
// 	IF snd_step = 0 THEN
// 		snd_text := CONCAT('Content-Type: application/octet-stream; name="',str2);
// 		step := 440;
// 	END_IF;
//
// 440:
// 	IF snd_step = 0 THEN
// 		snd_enable := TRUE;
// 		snd_text := CONCAT('Content-Disposition: attachment; filename="',str2);
// 		snd_lf_cnt := 2;
// 		step := 450;
// 	END_IF;
//
// 450:
// 	IF snd_step = 0 THEN
// 		FSD.FILENAME := str1; (* file name *)
// 		FSD.OFFSET := UDINT#0; (* start at beginning of file *)
// 		step := 460;
// 	END_IF;
//
// 460:
// 	FSD.MODE := BYTE#1; (* open existing file for reading *)
// 	F_BUF.SIZE := b64_max; (* read maximum length *)
// 	idx1 := 0;
// 	idx2 := 0;
// 	step := 470;
//
// 470:
// 	IF FSD.MODE = BYTE#0 AND FSD.ERROR = BYTE#0 THEN
// 		last_block := FSD.FILE_SIZE = FSD.OFFSET;
// 		b64_size1 := MIN(48,UINT_TO_INT(F_BUF.SIZE) - idx1);
// 		IF b64_size1 > 0 THEN
// 			idx3 := b64_size1 - 1;
// 			FOR i1 := 0 TO idx3 DO (* copy data into BASE64 buffer *)
// 				b64_buf1[i1] := F_BUF.BUFFER[idx1];
// 				idx1 := idx1 + 1;
// 			END_FOR;
// 			BASE64_ENCODE_STREAM( SIZE1:= b64_size1, BUF1:= b64_buf1, BUF2:= b64_buf2, SIZE2=> b64_size2); (* BASE64 encoding *)
// 			idx3 := b64_size2 - 1;
// 			FOR i1 := 0 TO idx3 DO (* copy data out of BASE64 buffer *)
// 				S_BUF.BUFFER[idx2] := b64_buf2[i1];
// 				idx2 := idx2 + 1;
// 			END_FOR;
// 			b64_lf := TRUE;
// 			(*####################  DEBUG-MESSAGE  ###################################*)
// 			(*IF _debug_enable THEN
// 				LOG_CL.NEW_MSG := 'B64: FILE ~1 /SIZE ~2 /OFF ~3 /BSIZE ~4 /idx1 ~5 /idx2 ~6';
// 				LOG_CL.PRINTF[1] := FSD.FILENAME;
// 				LOG_CL.PRINTF[2] := UDINT_TO_STRING(FSD.FILE_SIZE);
// 				LOG_CL.PRINTF[3] := UDINT_TO_STRING(FSD.OFFSET);
// 				LOG_CL.PRINTF[4] := INT_TO_STRING(b64_size1);
// 				LOG_CL.PRINTF[5] := INT_TO_STRING(idx1);
// 				LOG_CL.PRINTF[6] := INT_TO_STRING(idx2);
// 				LOG_MSG();
// 			END_IF;*)
// 			(*########################################################################*)
// 		ELSE
// 			b64_lf := last_block;
// 			step := 480; (* block finished  *)
// 		END_IF;
// 		IF b64_lf THEN
// 			S_BUF.BUFFER[idx2] := BYTE#16#0D;
// 			idx2 := idx2 + 1;
// 			S_BUF.BUFFER[idx2] := BYTE#16#0A;
// 			idx2 := idx2 + 1;
// 		END_IF;
// 		(*####################  DEBUG-MESSAGE  ###################################*)
// 		(*IF _debug_enable THEN
// 			LOG_CL.NEW_MSG := 'B64: exit ~1 /SIZE ~2 /OFF ~3 /eof ~4 /lf_cnt ~5';
// 			LOG_CL.PRINTF[1] := FSD.FILENAME;
// 			LOG_CL.PRINTF[2] := UDINT_TO_STRING(FSD.FILE_SIZE);
// 			LOG_CL.PRINTF[3] := UDINT_TO_STRING(FSD.OFFSET);
// 			LOG_CL.PRINTF[4] := BOOL_TO_STRING(last_block);
// 			LOG_CL.PRINTF[5] := INT_TO_STRING(snd_lf_cnt);
// 			LOG_MSG();
// 		END_IF;*)
// 		(*########################################################################*)
// 	END_IF;
//
// 480:
// 	S_BUF.SIZE := INT_TO_UINT(idx2); (* send data *)
// 	(*####################  DEBUG-MESSAGE  ###################################*)
// 	(*IF _debug_enable THEN
// 		LOG_CL.NEW_MSG := 'B64: tcp_send ~1';
// 		LOG_CL.PRINTF[1] := INT_TO_STRING(idx2);
// 		LOG_MSG();
// 	END_IF;*)
// 	(*########################################################################*)
// 	step := 490;
//
// 490:
// 	IF S_BUF.SIZE = UINT#0 THEN (* wait until all data is sent *)
// 		step := SEL(last_block ,460,400);
// 	END_IF;
//
// (* ++++++++++++++++++++++++++++++++++++++++ *)
//
// 800:
// 	IF snd_step = 0 THEN
// 		snd_enable := FALSE;
// 		snd_text := '--x--';
// 		snd_lf_cnt := 2;
// 		step := 810;
// 	END_IF;
//
// 810:
// 	IF snd_step = 0 THEN
// 		snd_enable := TRUE;
// 		snd_text := '.';
// 		snd_lf_cnt := 1;
// 		step := 820;
// 	END_IF;
//
// 820:
// 	IF rcv_state = 250 THEN (* 250 = Requested mail action okay *)
// 		snd_text := 'QUIT';
// 		ip_c_red_disable := TRUE;
// 		next_step := 830;
// 	END_IF;
//
// 830:
// 	IF rcv_state = 221  OR TON_WAIT.ET > timeout3 THEN (* 221 = Service closing transmission channel *)
// 		step := 900;
// 	END_IF;
//
// (* ================================================== *)
//
// 900:
// 	IF FILE_DELETE THEN (* delete files after transfer *)
// 		cnt1 := ELEMENT_COUNT(59, FILES) - 1; (* separator >;<, number of files *)
// 		step := 910;
// 	ELSE
// 		step := 950;
// 	END_IF;
//
// 910:
// 	IF FSD.MODE = BYTE#0 AND FSD.ERROR = BYTE#0 THEN
// 		IF cnt1 >= 0 THEN
// 			str1 := ELEMENT_GET(59, cnt1, FILES); (* separator >;< *)
// 			IF str1 <> '#DEL#' THEN
// 				FSD.FILENAME := str1;
// 				FSD.MODE := BYTE#4; (* File Remove *)
// 			END_IF;
// 			cnt1 := cnt1 - 1;
// 		ELSE
// 			step := 950;
// 		END_IF;
// 	END_IF;
//
// 950:
// 	DONE := TRUE;
// 	step := 980;
//
// 980:
// 	IP_C.C_ENABLE := FALSE; (* close SMTP control channel *)
// 	S_BUF.SIZE := UINT#0;
// 	R_BUF.SIZE := UINT#0;
// 	IP_C.MAILBOX[3] := BYTE#0; (* re-enable IP receive *)
// 	snd_step := 0;
// 	next_step := 0;
// 	FSD.MODE := BYTE#5; (* close file *)
// 	step := 990;
//
// 990:
// 	IF IP_C.C_STATE = BYTE#0 AND FSD.FILE_OPEN = FALSE THEN
// 		step := 0;
// 	END_IF;
//
// (*  +++++++++++++++++ authentication +++++++++++++++++ *)
//
// (* PLAIN ++++++++++++++++++++++++++++++++++++++++++++++++++++++++++ *)
//
// 1000:
// 	snd_text := CONCAT('AUTH',str3);
// 	snd_lf_cnt := 1;
//  	step := 1010;
//
// 1010:
// 	IF rcv_state = 334 THEN (* 334 = authentication  *)
// 		cnt1 := LEN(URL_DATA.USER);
// 		cnt2 := LEN(URL_DATA.PASSWORD);
// 		IF cnt1 + cnt2 <= 46 THEN (* USER + PASSWORD together may have at most 46 characters *)
// 			b64_buf1[0] := BYTE#0;
// 			FOR i1 := 1 TO cnt1 DO
// 				b64_buf1[i1] := CODE(URL_DATA.USER, i1);
// 			END_FOR;
// 			b64_size1 := cnt1 + 1;
// 			b64_buf1[b64_size1] := BYTE#0;
// 			b64_size1 := b64_size1 + 1;
// 			FOR i1 := 1 TO cnt2 DO
// 				b64_buf1[b64_size1] := CODE(URL_DATA.PASSWORD, i1);
// 				b64_size1 := b64_size1 + 1;
// 			END_FOR;
// 			BASE64_ENCODE_STREAM( SIZE1:= b64_size1, BUF1:= b64_buf1, BUF2:= b64_buf2, SIZE2=> b64_size2); (* BASE64 encoding *)
// 			idx1 := b64_size2 - 1;
// 			FOR i1 := 0 TO idx1 DO
// 				S_BUF.BUFFER[i1] := b64_buf2[i1];
// 			END_FOR;
// 			S_BUF.BUFFER[b64_size2] := BYTE#16#0D;
// 			b64_size2 := b64_size2 + 1;
// 			S_BUF.BUFFER[b64_size2] := BYTE#16#0A;
// 			b64_size2 := b64_size2 + 1;
// 			S_BUF.SIZE := INT_TO_UINT(b64_size2);
// 			rcv_state := 0;
// 		END_IF;
// 		step := 90;
// 	END_IF;
//
// (* LOGIN ++++++++++++++++++++++++++++++++++++++++++++++++++++++++++ *)
//
// 1100:
// 	snd_text := CONCAT('AUTH',str3);
// 	snd_lf_cnt := 1;
//  	step := 1110;
//
// 1110:
// 	IF rcv_state = 334 THEN (* 334 = authentication  *)
// 		b64_str1 := URL_DATA.USER;
// 		b64_start := TRUE; (* BASE64 encoding of username *)
// 		step := 1120;
// 	END_IF;
//
// 1120:
// 	IF b64_start AND b64_done THEN
// 		b64_start := FALSE;
// 		snd_text := b64_str2;
// 		next_step := 1130;
// 	END_IF;
//
// 1130:
// 	IF rcv_state = 334 THEN (* 334 = Password:  *)
// 		b64_str1 := URL_DATA.PASSWORD;
// 		b64_start := TRUE; (* BASE64 encoding of password *)
// 		step := 1140;
// 	END_IF;
//
// 1140:
// 	IF b64_start AND b64_done THEN
// 		b64_start := FALSE;
// 		snd_text := b64_str2;
// 		next_step := 90;
// 	END_IF;
//
// (* CRAM-MD5  ++++++++++++++++++++++++++++++++++++++++++++++++++++++++++
// (Challenge-Response Authentication Mechanism, Message Digest 5) authentication based on the MD5-HMAC algorithm. *)
//
// 1200:
// 	snd_text := CONCAT('AUTH',str3);
// 	snd_lf_cnt := 1;
//  	step := 1210;
//
// 1210:
// 	IF rcv_state = 334 THEN (* 334 = authentication  *)
// 		md5_b64_ts := RIGHT(rcv_text,LEN(rcv_text) - 4);
// 		md5_user := URL_DATA.USER;
// 		md5_password := URL_DATA.PASSWORD;
// 		MD5_RUN := TRUE;
// 		step := 1220;
// 	END_IF;
//
// 1220:
// 	MD5_CRAM_AUTH(RUN:=MD5_RUN,USERNAME:=md5_user,PASSWORD:=md5_password,B64_TS:=md5_b64_ts,AUTH_KEY:=md5_auth_key);
// 	IF NOT MD5_RUN THEN
// 		snd_text := md5_auth_key;
// 		step := 90;
// 	END_IF;
//
// (* STARTTLS  ++++++++++++++++++++++++++++++++++++++++++++++++++++++++++ *)
//
// 1300:
// 	snd_text := 'STARTTLS';
// 	snd_lf_cnt := 1;
//  	step := 1310;
//
// 1310:
// 	IF rcv_state = 220 THEN (* 220 = Service ready - Ready to start TLS *)
// 		IP_C.MAILBOX[16] := BYTE#1; (* activate SSL/TLS *)
// 		step := 1320;
// 	END_IF;
//
// 1320:
// 	IF IP_C.MAILBOX[16] = BYTE#2 THEN (* wait until SSL/TLS has been activated *)
// 		step := 30; (* restart the whole sequence from the beginning *)
// 	END_IF;
//
// (* no authentication found +++++++++++++++++++++++++++++++ *)
// 1900: ; (* wait for runtime error *)
//
// END_CASE;
// (* ++++++++++++++++++++++++++++++++++++++++++++++++++++++++++ *)
// IF step >= 30 THEN
// 	IF R_BUF.SIZE > UINT#0 THEN (* data received? *)
// 		idx1 := UINT_TO_INT(R_BUF.SIZE);
// 		REPEAT (* detect line termination and determine real end of TEXT *)
// 			idx1 := idx1 - 1;
// 		UNTIL idx1 = 0 OR R_BUF.BUFFER[idx1] >= BYTE#32 (* TRUE = EXIT *)
// 		END_REPEAT;
// 		FOR i1 := 0 TO idx1 DO (* for multiline replace all CRLF with >^< *)
// 			IF R_BUF.BUFFER[i1] < BYTE#32 THEN
// 				R_BUF.BUFFER[i1] := BYTE#94; (* >^< *)
// 			END_IF;
// 		END_FOR;
// 		rcv_text := BUFFER_TO_STRING(PT:=REF(R_BUF.BUFFER),SIZE:=idx1+1,START:=0,STOP:=STRING_LENGTH-1);
// 		IF LEN(rcv_text) >= 3 THEN (* check and evaluate status code *)
// 			rcv_s := LEFT(rcv_text,3);
// 			IF IS_NUM(STR:=rcv_s) THEN (* contains only digits? *)
// 				rcv_state := STRING_TO_INT(rcv_s);
// 			END_IF;
// 			IP_C.R_OBSERVE := FALSE;
// 		END_IF;
// 		R_BUF.SIZE := UINT#0; (* delete data *)
//
// 		(*####################  DEBUG-MESSAGE  ###################################*)
// 		(*IF _debug_enable THEN
// 			LOG_CL.NEW_MSG := 'RCV: >~1<';
// 			LOG_CL.PRINTF[1] := rcv_text;
// 			LOG_MSG();
// 		END_IF;*)
// 		(*########################################################################*)
//
// 	END_IF;
// END_IF;
//
// (* automatic data sending *)
//
// CASE snd_step OF
//
// 00:
// 	IF LEN(snd_text) > 0 THEN
//
// 		(*####################  DEBUG-MESSAGE  ###################################*)
// 		(*IF _debug_enable THEN
// 			LOG_CL.NEW_MSG := 'SND: >~1< /lf ~2';
// 			LOG_CL.PRINTF[1] := snd_text;
// 			LOG_CL.PRINTF[2] := INT_TO_STRING(snd_lf_cnt);
// 			LOG_MSG();
// 		END_IF;*)
// 		(*########################################################################*)
//
// 		_STRING_TO_BUFFER(str:=snd_text,pos:=snd_idx,pt:=REF(S_BUF.BUFFER),size:=SIZEOF(S_BUF.BUFFER)); (* copy string into buffer *)
// 		snd_idx := snd_idx + LEN(snd_text);
// 		FOR i1 := 1 TO snd_lf_cnt DO
// 			S_BUF.BUFFER[snd_idx] := BYTE#16#0D;
// 			snd_idx := snd_idx + 1;
// 			S_BUF.BUFFER[snd_idx] := BYTE#16#0A;
// 			snd_idx := snd_idx + 1;
// 		END_FOR;
// 		snd_text := '';
// 		rcv_state := 9999; (* clear last SMTP status *)
//
// 		IF snd_enable THEN
// 			S_BUF.SIZE := INT_TO_UINT(snd_idx); (* enter send length *)
// 			R_BUF.SIZE := UINT#0; (* reset receive buffer *)
// 			IP_C.R_OBSERVE := step <= 120 OR step >= 820;
// 			snd_idx := 0;
// 			snd_step := 10;
// 		END_IF;
// 	END_IF;
//
// 10:
// 	IF S_BUF.SIZE = UINT#0 THEN (* wait until all data is sent *)
// 		IF next_step <> 0 THEN
// 			step := next_step;
// 			next_step := 0;
// 		END_IF;
// 		snd_step := 0;
// 	END_IF;
//
// END_CASE;
//
// (* global error handling for main routine *)
// IF ERROR_T = BYTE#0 AND step > 20 THEN (* no error stored yet and main routine active *)
//
// 	IF IP_C.ERROR > DWORD#0 AND IP_C.C_ENABLE AND NOT IP_C.TIME_RESET THEN  (* IP Control 1 *)
// 		IF ip_c_red_disable = FALSE OR IP_C.ERROR <> DWORD#16#FD000000 THEN
// 			ERROR_C := IP_C.ERROR;
// 			ERROR_T := BYTE#2;
// 			step := 980;
// 		END_IF;
// 	END_IF;
//
// 	IF FSD.MODE = BYTE#0 THEN
// 		IF FSD.ERROR > BYTE#0 THEN
// 			ERROR_C := BYTE_TO_DWORD(FSD.ERROR);
// 			ERROR_T := BYTE#4; (* file access *)
// 			step := 980;
// 		END_IF;
// 	END_IF;
// END_IF;
//
// IF TON_WAIT.Q THEN (* sequence fault - step chain *)
// 	ERROR_C := SHL(INT_TO_DWORD(step),16) OR INT_TO_DWORD(rcv_state); (* enter current step and last SMTP status *)
// 	ERROR_T := BYTE#5;
// 	step := 980;
// END_IF;
//
// (* ######################################################## *)
//
// DNS_CLIENT(IP_C:=IP_C, S_BUF:=S_BUF, R_BUF:=R_BUF, DOMAIN:=URL_DATA.DOMAIN, IP4_DNS:= DNS_IP4, ACTIVATE:=step=10); (* DNS-Client *)
// IPC(IP:= DWORD#0, PORT:= WORD#0 , TIME_OUT:= TIMEOUT, IP_C:= IP_C, S_BUF:= S_BUF, R_BUF:= R_BUF); (* SMTP control channel *)
// FS(FSD:=FSD,PT:=F_BUF); (* FILE_SERVER *)
// BASE64_ENCODE_STR(RUN:= b64_start, STR1:= b64_str1, STR2:= b64_str2, DONE=> b64_done); (* BASE64 encoding *)
//
// TON_WAIT(IN:=step = last_step AND step > 0,PT:=timeout2);
// last_step := step;
// activate_last := ACTIVATE;
// BUSY := step <> 0;
// END_FUNCTION_BLOCK

FUNCTION_BLOCK SNTP_CLIENT
VAR_IN_OUT
	IP_C : IP_C; (* IP_Control management structure *)
	S_BUF : NETWORK_BUFFER;
	R_BUF : NETWORK_BUFFER;
END_VAR
VAR_INPUT
	IP4 : DWORD;
	ACTIVATE : BOOL;
END_VAR
VAR_OUTPUT
	ERROR : DWORD;
	DONE_P : BOOL;
	UDT : DT;
	XMS : INT;
END_VAR
VAR
	IP_FIFO : IP_FIFO;
	ip_state : BYTE;
	ip_id : BYTE;
	i : INT;
	last : DWORD;
	state : INT;
	tx : DWORD;
	activate_last : BOOL;
	ip4_stored : DWORD;

END_VAR

(* Domain Name System (query) *)
tx := T_PLC_MS(); (* read system time *)

CASE state OF
00: (* wait for rising edge on SET *)
	DONE_P := FALSE;
	IF ACTIVATE AND NOT activate_last THEN
		ip4_stored := IP4; (* store current IP4 *)
		state := 10;
		ERROR := DWORD#0;
		ip_state := BYTE#1; (* register *)
		(*####################  DEBUG-MESSAGE  ###################################*)
		(*########################################################################*)
	END_IF;

10: (* register with IP_Control and wait for release *)
	IF ip_state = BYTE#3 THEN

		S_BUF.BUFFER[00] := BYTE#16#1B;
		FOR i := 1 TO 47 DO
			S_BUF.BUFFER[i] := BYTE#16#00;
		END_FOR;

		last := tx; (* save current time value *)
		state := 30;

		(* set up IP data traffic *)
		IP_C.C_PORT := WORD#123; (* enter port number *)
		IP_C.C_IP := ip4_stored; (* enter IP *)
		IP_C.C_MODE := BYTE#1; (* Mode: UDP+ACTIVE+PORT+IP *)
		IP_C.C_ENABLE := TRUE; (* enable connection setup *)
		IP_C.TIME_RESET := TRUE; (* reset timeout monitoring *)
		IP_C.R_OBSERVE := TRUE; (* monitor data reception *)
		S_BUF.SIZE := UINT#48; (* enter send length *)
		R_BUF.SIZE := UINT#0; (* reset receive length *)
    		(*####################  DEBUG-MESSAGE  ###################################*)
    		(*########################################################################*)
	END_IF;

30:
	IF IP_C.ERROR <> DWORD#00 THEN
		ERROR := IP_C.ERROR;
		S_BUF.SIZE := UINT#0;
		R_BUF.SIZE := UINT#0;
		state := 0;
    		(*####################  DEBUG-MESSAGE  ###################################*)
    		(*########################################################################*)

	ELSIF S_BUF.SIZE = UINT#0 AND R_BUF.SIZE >= UINT#48 THEN (* check length of received data *)

		(* convert SNTP timestamp base 1900-01-01 -> Unix 1970-01-01 = +2208988800 seconds*)
		UDT := DWORD_TO_DT(DWORD_OF_BYTE(R_BUF.BUFFER[40],R_BUF.BUFFER[41],R_BUF.BUFFER[42],R_BUF.BUFFER[43]) - DWORD#2208988800);

		(* original fractional seconds are represented as a 32 bit fraction *)
		(* calculate ms only with reduced resolution 1/65535 -> use high word *)
		XMS := DWORD_TO_INT(SHR(DINT_TO_DWORD(WORD_TO_DINT(WORD_OF_BYTE(R_BUF.BUFFER[44],R_BUF.BUFFER[45])) * DINT#1000),16));
		(* divide the time difference (runtime error) between send and receive by 2 and add *)
		XMS := XMS + DWORD_TO_INT(SHR(tx - last,1));

		UDT := DWORD_TO_DT(DT_TO_DWORD(UDT) + (XMS / 1000)); (* add the fractional seconds of the time difference to UDT *)
		XMS := XMS MOD 1000;  (* take over ms *)
		state := 0;
		DONE_P := TRUE;
    		(*####################  DEBUG-MESSAGE  ###################################*)
    		(*########################################################################*)

	END_IF;

	IF state = 0 THEN
		IP_C.R_OBSERVE := FALSE; (* monitor data reception *)
		ip_state := BYTE#4;
	END_IF;

END_CASE;

activate_last := ACTIVATE; (* save last status for edge detection *)

(* IP_FIFO *)
IP_FIFO(FIFO:=IP_C.FIFO,STATE:=ip_state,ID:=ip_id);

(***************************************************************************************)
END_FUNCTION_BLOCK

FUNCTION_BLOCK SNTP_SERVER
VAR_IN_OUT
	IP_C : IP_C; (* IP_Control management structure *)
	S_BUF : NETWORK_BUFFER;
	R_BUF : NETWORK_BUFFER;
END_VAR
VAR_INPUT
	ENABLE : BOOL;
	STRATUM : BYTE := BYTE#1;
	UDT : DT;
	XMS : INT;
END_VAR
VAR
	IP_FIFO : IP_FIFO;
	ip_state : BYTE;
	ip_id : BYTE;
	i2 : INT;
	i : INT;
	timestamp_int : DWORD; (* Timestamp integer part *)
	timestamp_sek : DWORD; (* Timestamp fraction part (HIGH_WORD) *)
	ts_b : BYTE;
	state : INT;
	tx : UDINT;
	t : TON;

END_VAR

(* Domain Name System (query) *)
tx := T_PLC_MS(); (* read system time *)

CASE state OF

00: (* wait for release *)
	IF ENABLE THEN
		state := 10;
		ip_state := BYTE#1; (* register *)
    		(*####################  DEBUG-MESSAGE  ###################################*)
    		(*########################################################################*)
	END_IF;

10: (* register with IP_Control and wait for release *)
	IF ip_state = BYTE#3 THEN
		(* set up IP data traffic *)
		IP_C.C_PORT := WORD#123; (* enter port number *)
		IP_C.C_IP := DWORD#00; (* enter IP *)
		IP_C.C_MODE := BYTE#5; (* Mode: UDP+PASSIV+PORT *)
		IP_C.C_ENABLE := TRUE; (* enable connection setup *)
		IP_C.TIME_RESET := TRUE; (* reset timeout monitoring *)
		IP_C.R_OBSERVE := FALSE; (* monitor data reception *)
		S_BUF.SIZE := UINT#0; (* enter send length *)
		R_BUF.SIZE := UINT#0; (* reset receive length *)
		state := 20;
    		(*####################  DEBUG-MESSAGE  ###################################*)
    		(*########################################################################*)
	END_IF;
20:
	IF R_BUF.SIZE > UINT#0 THEN
		state := 20;
    		(*####################  DEBUG-MESSAGE  ###################################*)
    		(*########################################################################*)
		(* pad received telegram with 00 if too short! and preset send buffer with 00 *)
		FOR i := 0 TO 47 DO
			IF INT_TO_UINT(i) > R_BUF.SIZE - 1 THEN
				R_BUF.BUFFER[i] := BYTE#00;
			END_IF;
			S_BUF.BUFFER[i] := BYTE#00;
		END_FOR;

		R_BUF.SIZE := UINT#0;

		(* prepare send data *)
		S_BUF.BUFFER[0] := BYTE#2#11100; (* Flags: NO WARNING, NTP VERSION 3 , SERVER *)
		S_BUF.BUFFER[1] := STRATUM; (* Peer Clock Stratum: *)
		S_BUF.BUFFER[2] := BYTE#10; (* peer polling interval 2 to the power of 10 = 1024 sec. *)
		S_BUF.BUFFER[3] := BYTE#16#FB; (* Peer Clock Precision: -5 = -31,25ms *)

		(* convert SNTP timestamp base 1900-01-01 = Unix 1970-01-01 + 2208988800 seconds *)
		timestamp_int := DT_TO_DWORD(UDT) + DWORD#2208988800;

		(* fractional seconds are represented as a 32 bit fraction *)
		(* calculate only with reduced resolution 1/65535 -> use high word *)
		(* calculation of the fractional seconds: xms * 65535 / 1000 *)
		timestamp_sek := DINT_TO_DWORD(DWORD_TO_DINT(SHL(INT_TO_DWORD(XMS),16))/DINT#1000);

		ts_b := BYTE_OF_DWORD(timestamp_int,3); (* Timestamp Byte 3 *)
		S_BUF.BUFFER[16] := ts_b; (* Reference Timestamp *)
		S_BUF.BUFFER[32] := ts_b; (* Receive   Timestamp *)
		S_BUF.BUFFER[40] := ts_b; (* Transmit  Timestamp *)

		ts_b := BYTE_OF_DWORD(TIMESTAMP_INT,2); (* Timestamp Byte 2 *)
		S_BUF.BUFFER[17] := ts_b; (* Reference Timestamp *)
		S_BUF.BUFFER[33] := ts_b; (* Receive   Timestamp *)
		S_BUF.BUFFER[41] := ts_b; (* Transmit  Timestamp *)

		ts_b := BYTE_OF_DWORD(TIMESTAMP_INT,1); (* Timestamp Byte 1 *)
		S_BUF.BUFFER[18] := ts_b; (* Reference Timestamp *)
		S_BUF.BUFFER[34] := ts_b; (* Receive   Timestamp *)
		S_BUF.BUFFER[42] := ts_b; (* Transmit  Timestamp *)

		ts_b := BYTE_OF_DWORD(TIMESTAMP_INT,0); (* Timestamp Byte 0 *)
		S_BUF.BUFFER[19] := ts_b; (* Reference Timestamp *)
		S_BUF.BUFFER[35] := ts_b; (* Receive   Timestamp *)
		S_BUF.BUFFER[43] := ts_b; (* Transmit  Timestamp *)

		ts_b := BYTE_OF_DWORD(TIMESTAMP_SEK,1); (* Timestamp Byte 1 *)
		S_BUF.BUFFER[20] := ts_b; (* Reference Timestamp *)
		S_BUF.BUFFER[36] := ts_b; (* Receive   Timestamp *)
		S_BUF.BUFFER[44] := ts_b; (* Transmit  Timestamp *)

		ts_b := BYTE_OF_DWORD(timestamp_sek,0);	(* Timestamp Byte 0 *)
		S_BUF.BUFFER[21] := ts_b; (* Reference Timestamp *)
		S_BUF.BUFFER[37] := ts_b; (* Receive   Timestamp *)
		S_BUF.BUFFER[45] := ts_b; (* Transmit  Timestamp *)

		(* copy bytes 1-8 of transmit time to originate time *)
		i2 := 40;
		FOR i := 24 TO 31 DO
			S_BUF.BUFFER[i] := R_BUF.BUFFER[i2];
			i2 := i2 +1;
		END_FOR;

		S_BUF.SIZE := UINT#48; (* send data *)

	ELSIF NOT ENABLE AND S_BUF.SIZE = UINT#0 THEN
		ip_state := BYTE#4; (* unregister *)
		state := 0;
	END_IF;

END_CASE;

t(IN:= IP_C.ERROR > DWORD#0, PT:=T#5s);
IF t.Q THEN
  IP_C.TIME_RESET := TRUE; (* Error Reset *)
END_IF;

(* IP_FIFO *)
IP_FIFO(FIFO:=IP_C.FIFO,STATE:=ip_state,ID:=ip_id);
END_FUNCTION_BLOCK

// Commented out for beedance: it uses BUFFER_TO_STRING, which is commented out.
// FUNCTION_BLOCK SPIDER_ACCESS
// VAR_IN_OUT
// 	IP_C : IP_C;(*IP_Control management structure*)
// 	S_BUF : NETWORK_BUFFER;
// 	R_BUF : NETWORK_BUFFER;
// 	VALUE : STRING;
// 	VAR_NAME : STRING(40);
// END_VAR
// VAR_INPUT
// 	MODE : BYTE;
// END_VAR
// VAR_OUTPUT
// 	ERROR : DWORD;
// END_VAR
// VAR
// 	state : INT;
// 	st_tmp : STRING(STRING_LENGTH);
// 	URL_DATA : url;
// 	HTTP_GET : HTTP_GET;
// 	value_len :	UINT;
// 	body_len :	UINT;
// 	mode_save : BYTE;
// END_VAR
//
// CASE state OF
//
// 00:
// 	IF MODE > BYTE#0 AND MODE < BYTE#3 THEN
// 		MODE_SAVE := MODE; (* store mode *)
// 		(* if there is no '.' in the name, it is a global variable *)
// 		IF FIND(VAR_NAME,'.') = 0 THEN
// 			st_tmp := CONCAT('%40GV.',VAR_NAME);
// 		ELSE
// 			st_tmp := VAR_NAME;
// 		END_IF;
//
// 		IF MODE_SAVE = BYTE#2 THEN (* 2 = Write *)
// 			VALUE_LEN := INT_TO_UINT(LEN(VALUE));
// 			st_tmp := CONCAT(st_tmp,'+');
// 			st_tmp := CONCAT(st_tmp,VALUE);
// 			URL_DATA:=STRING_TO_URL(STR:= CONCAT('http://x/dir/cgi-bin/writeVal.exe?',st_tmp),DEFAULT_PROTOCOL:='',DEFAULT_PATH:='');
// 		ELSE
// 			URL_DATA:=STRING_TO_URL(STR:= CONCAT('http://x/dir/cgi-bin/readVal.exe?',st_tmp),DEFAULT_PROTOCOL:='',DEFAULT_PATH:='');
// 		END_IF;
//
// 		state := 60;
// 	END_IF;
// 60:
// 	IF HTTP_GET.DONE THEN
// 		IF MODE_SAVE = BYTE#2 THEN (* Write *)
// 			BODY_LEN := HTTP_GET.BODY_STOP - HTTP_GET.BODY_START + BOOL_TO_UINT(HTTP_GET.BODY_STOP > UINT#0);
// 			ERROR := BOOL_TO_DWORD(BODY_LEN <> VALUE_LEN);
// 		ELSE (* Read *)
// 			IF HTTP_GET.BODY_START > 0 THEN
// 				VALUE := BUFFER_TO_STRING(PT:=REF(R_BUF.BUFFER),SIZE:=R_BUF.SIZE,START:=UINT_TO_INT(HTTP_GET.BODY_START),STOP:=UINT_TO_INT(HTTP_GET.BODY_STOP));
// 			ELSE
// 				VALUE := '';
// 			END_IF;
// 		END_IF;
// 		STATE   := 100;
//
// 	ELSIF (HTTP_GET.ERROR > DWORD#00) THEN
// 		ERROR := HTTP_GET.ERROR;
// 		STATE   := 100;
// 	END_IF;
//
// 100:
// 	(* UNLOCK HTTP DATA *)
// 	IF HTTP_GET.DONE = FALSE THEN
// 		STATE := 0;
// 	END_IF;
//
// END_CASE;
//
// (* HTTP_GET *)
// HTTP_GET(	IP_C:=IP_C,
// 			S_BUF:=S_BUF,
// 			R_BUF:=R_BUF,
// 			IP4:=DWORD#00,
// 			GET:=state=60,
// 			MODE:=BYTE#0,
// 			UNLOCK_BUF:=state=100,
// 			URL_DATA:=URL_DATA
// 			);
// END_FUNCTION_BLOCK

FUNCTION STRING_TO_URL : URL
VAR_INPUT
	STR : STRING(STRING_LENGTH);
	DEFAULT_PROTOCOL : STRING(10);
	DEFAULT_PATH : STRING(80);
END_VAR
VAR
	pos: INT;
	pos2: INT;
	x : STRING(STRING_LENGTH);
END_VAR

(* check if string is empty and return empty url *)
IF STR = '' THEN RETURN; END_IF;

(* extract the protocol *)
(* first we check if the optional protocol is specified ending with a :// *)
pos := FIND(STR, '://');
IF pos > 0 THEN
	(* store protocol and restore the rest of url in temp *)
	STRING_TO_URL.PROTOCOL := LEFT(STR, pos - 1);
	x := RIGHT(STR, LEN(STR) - pos - 2);
ELSE
	x := STR;
	STRING_TO_URL.PROTOCOL := DEFAULT_PROTOCOL;
END_IF;

(* extract user and password if present ending with a @ *)
pos := FINDB(STR1:=x,STR2:='@'); (* Find last @ *)

IF pos > 0 THEN
	(* extract user *)
	pos2 := FIND(x,':')+1;
	IF pos2 > 1 AND pos2 <= pos THEN
		STRING_TO_URL.USER := LEFT(x,pos2 - 2);
		STRING_TO_URL.PASSWORD := MID(x, pos - pos2, pos2);
	ELSE
		STRING_TO_URL.USER := LEFT(x, pos - 2);
		STRING_TO_URL.PASSWORD := '';
	END_IF;
	x := RIGHT(x, LEN(x) - pos);
ELSE
	STRING_TO_URL.USER := '';
	STRING_TO_URL.PASSWORD := '';
END_IF;

(* extract anchor *)
pos := FIND(x, '#');
IF pos > 0 THEN
	STRING_TO_URL.ANCHOR := RIGHT(x, LEN(x) - pos);
	x := LEFT(x, pos - 1);
ELSE
	STRING_TO_URL.ANCHOR := '';
END_IF;

(* extract query  *)
pos := FIND(x, '?');
IF pos > 0 THEN
	STRING_TO_URL.QUERY := RIGHT(x, LEN(x) - pos);
	x := LEFT(x, pos - 1);
ELSE
	STRING_TO_URL.QUERY := '';
END_IF;

(* extract path  *)
pos := FIND(x, '/');
IF pos > 0 THEN
	STRING_TO_URL.PATH := RIGHT(x, LEN(x) - pos + 1);
	x := LEFT(x, pos - 1);
ELSE
	STRING_TO_URL.PATH := DEFAULT_PATH;
END_IF;

(* extract port and leave domain *)
pos := FIND(x, ':');
IF pos > 0 THEN
	STRING_TO_URL.PORT := STRING_TO_WORD(RIGHT(x, LEN(x) - pos));
	STRING_TO_URL.DOMAIN := LEFT(x, pos - 1);
ELSE
	STRING_TO_URL.PORT := 0;
	STRING_TO_URL.DOMAIN := x;
END_IF;
END_FUNCTION

// Commented out for beedance: it uses DT_TO_STRF, which is commented out.
// FUNCTION_BLOCK SYS_LOG
// VAR_IN_OUT
// 	IP_C : IP_C; (* IP_Control management structure *)
// 	S_BUF : NETWORK_BUFFER;
// 	R_BUF : NETWORK_BUFFER;
// END_VAR
// VAR_INPUT
// 	ACTIVATE : BOOL;
// 	LDT : DT;
// 	SERVER_IP4 : DWORD;
// 	PORT : WORD;
// 	FACILITY : BYTE;
// 	SEVERITY : BYTE;
// 	TAG : STRING(32);
// 	HOSTNAME : STRING;
// 	MESSAGE : STRING(STRING_LENGTH);
// 	OPTION : BYTE;
// END_VAR
// VAR_OUTPUT
// 	DONE_P : BOOL;
// 	ERROR : DWORD;
// END_VAR
// VAR
// 	ip_state : BYTE;
// 	ip_id : BYTE;
// 	IP_FIFO : IP_FIFO;
// 	activate_last : BOOL;
// 	state : INT;
// 	s1 : STRING(20);
// 	i : INT;
//
// 	(*LOG_MSG : LOG_MSG;
// 	_debug_enable : BOOL := TRUE;*)
//
// END_VAR
//
// CASE state OF
// 00: (* wait for rising edge on SET *)
// 	IF ACTIVATE AND NOT ACTIVATE_LAST THEN
// 		state := 10;
// 		ERROR := DWORD#0;
// 		IP_STATE := BYTE#1; (* register *)
//     		(*####################  DEBUG-MESSAGE  ###################################*)
//     		(*IF _debug_enable THEN
//       			LOG_CL.NEW_MSG := 'SYS_LOG: S00 START /IP_ID ~4';
//       			LOG_CL.PRINTF[4]  := BYTE_TO_STRING(IP_ID);
//       			LOG_MSG();
//     		END_IF;*)
//     		(*########################################################################*)
// 	END_IF;
// 	DONE_P := FALSE;
//
// 10: (* register with IP_Control and wait for release *)
// 	IF IP_STATE = BYTE#3 THEN
// 		(* prepare send data *)
// 		i := 0;
// 		IF (OPTION AND BYTE#0000_0001) = BYTE#00 THEN (* Option: no priority Code *)
// 			(* Priority:  '<xx>' as decimal value *)
// 			(* BYTE: xxxx x...  = Facility *)
// 			(*       .... .xxx  = Level *)
// 			s1 := REPLACE('<P>',BYTE_TO_STRING(SHL(FACILITY,3) OR (SEVERITY AND BYTE#0000_0111)),1,2);
// 		ELSE
// 			s1 := '';
// 		END_IF;
//
// 		IF (OPTION AND BYTE#0000_0010) = BYTE#00 THEN (* Option: No Use Syslog RFC Header *)
// 			(* 'month day hh:mm:ss ' *)
// 			s1 := CONCAT(s1,DT_TO_STRF(DTI:=LDT,MS:=0,FMT:='#E #W #N:#R:#T ',LANG:=1));
// 			_STRING_TO_BUFFER(STR:=s1,POS:=i,PT:=REF(S_BUF.BUFFER),SIZE:=UINT#1024);
// 			i := i + LEN(s1);
// 			(* ' enter sourcename *)
// 			_STRING_TO_BUFFER(STR:=HOSTNAME,POS:=i,PT:=REF(S_BUF.BUFFER),SIZE:=UINT#1024);
// 			i := i + LEN(HOSTNAME);
// 			S_BUF.BUFFER[i] := BYTE#32; (* insert space *)
// 			i := i + 1;
// 			(* ' enter tag *)
// 			_STRING_TO_BUFFER(STR:=TAG,POS:=i,PT:=REF(S_BUF.BUFFER),SIZE:=UINT#1024);
// 			i := i + LEN(TAG);
// 			S_BUF.BUFFER[i] := BYTE#32; (* insert space *)
// 			i := i + 1;
// 		END_IF;
//
// 		(* ' enter message *)
// 		_STRING_TO_BUFFER(STR:=MESSAGE,POS:=i,PT:=REF(S_BUF.BUFFER),SIZE:=UINT#1024);
// 		i := i + LEN(MESSAGE);
//
// 		IF (OPTION AND BYTE#0000_0100) > BYTE#00 THEN (* Option: Add a CR & LF to end of message *)
// 			S_BUF.BUFFER[i] := BYTE#13; (* insert carriage return *)
// 			i := i + 1;
// 			S_BUF.BUFFER[i] := BYTE#10; (* insert line feed *)
// 			i := i + 1;
// 		END_IF;
//
// 		state := 30;
//
// 		(* set up IP data traffic *)
// 		IF (OPTION AND BYTE#2#0000_1000) > BYTE#00 THEN (* Option: TCP Mode *)
// 			IP_C.C_MODE := BYTE#0; (* Mode: TCP/ACTIVE *)
// 		ELSE
// 			IP_C.C_MODE := BYTE#1; (* Mode: UDP/ACTIVE *)
// 		END_IF;
//
// 		IF PORT = WORD#0 THEN (* no port number specified? *)
// 			IF IP_C.C_MODE = BYTE#0 THEN (* determine mode  TCP or UDP? *)
// 				IP_C.C_PORT := WORD#1468; (* default port number for syslog over TCP *)
// 			ELSE
// 				IP_C.C_PORT := WORD#514; (* default port number for syslog over UDP *)
// 			END_IF;
// 		ELSE
// 			IP_C.C_PORT := PORT; (* enter the given port number *)
// 		END_IF;
//
// 		IP_C.C_IP := SERVER_IP4; (* enter IP *)
// 		IP_C.C_ENABLE := TRUE; (* enable connection setup *)
// 		IP_C.TIME_RESET := TRUE; (* reset timeout monitoring *)
// 		IP_C.R_OBSERVE := FALSE; (* monitor data reception *)
// 		S_BUF.SIZE := INT_TO_UINT(i); (* enter send length *)
// 		R_BUF.SIZE := UINT#0; (* reset receive length *)
//     		(*####################  DEBUG-MESSAGE  ###################################*)
//     		(*IF _debug_enable THEN
//       			LOG_CL.NEW_MSG := 'SYS_LOG: S20 SEND /IP_ID ~4';
//       			LOG_CL.PRINTF[4]  := BYTE_TO_STRING(IP_ID);
//       			LOG_MSG();
//     		END_IF;*)
//     		(*########################################################################*)
// 	END_IF;
//
// 30:
// 	IF IP_C.ERROR <> DWORD#00 THEN
// 		ERROR := IP_C.ERROR;
// 		state := 0;
//     		(*####################  DEBUG-MESSAGE  ###################################*)
//     		(*IF _debug_enable THEN
//       			LOG_CL.NEW_MSG := 'SYS_LOG: S30 ERROR ~1 IP_ID ~4';
//       			LOG_CL.PRINTF[1]  := DWORD_TO_STRING(ERROR);
//       			LOG_CL.PRINTF[4]  := BYTE_TO_STRING(IP_ID);
//       			LOG_MSG();
//     		END_IF;*)
//     		(*########################################################################*)
// 	ELSIF S_BUF.SIZE = UINT#0 THEN (* wait until all data is sent *)
// 		DONE_P := TRUE;
// 		state := 0;
//     		(*####################  DEBUG-MESSAGE  ###################################*)
//     		(*IF _debug_enable THEN
//       			LOG_CL.NEW_MSG := 'SYS_LOG: S30 OK /IP_ID ~4';
//       			LOG_CL.PRINTF[4]  := BYTE_TO_STRING(IP_ID);
//       			LOG_MSG();
//     		END_IF;*)
//     		(*########################################################################*)
// 	END_IF;
//
// 	IF state = 0 THEN (* release connection *)
// 		IP_STATE := BYTE#4;
// 	END_IF;
//
// END_CASE;
//
// ACTIVATE_LAST := ACTIVATE; (* save last status for edge detection *)
//
// (* IP_FIFO *)
// IP_FIFO(FIFO:=IP_C.FIFO,STATE:=ip_state,ID:=IP_ID);
// END_FUNCTION_BLOCK

FUNCTION_BLOCK TELNET_LOG
VAR_IN_OUT
	IP_C : IP_C;
	S_BUF : NETWORK_BUFFER;
	LOG_CL : LOG_CONTROL;
END_VAR
VAR_INPUT
	ENABLE : BOOL;
	OPTION : BYTE := BYTE#2#1000_1100; (* no flush buffer (7) , CR&LF (3), Colors (2), AUTOWRAP (1), Screen-Init (0) *)
	PORT : WORD := 23; (* port number *)
END_VAR
VAR_OUTPUT
	READY : BOOL;
END_VAR
VAR
	TELNET_PRINT : TELNET_PRINT;
	done : BOOL;
	init : BOOL;
	watchdog : TON;
	ci : INT;
	pi : INT;
	pi_last : INT;
	send : BOOL;
END_VAR

IF NOT init THEN
	init := TRUE;
	IF OPTION > 0 THEN
		TELNET_PRINT.OPTION := OPTION;
	END_IF;
	IF PORT > 0 THEN (* a specified port overrides the default port *)
		TELNET_PRINT.PORT := PORT;
	END_IF;
  	WATCHDOG.PT := T#1ms;
END_IF;

WATCHDOG(IN:=FALSE); (* stop timer *)

ci := LOG_CL.IDX;

(* evaluate CONNECT_OFF edge *)
IF IP_C.C_STATE = BYTE#1 THEN
	pi := 0;
	init := FALSE;
END_IF;

REPEAT
	IF pi <> ci AND IP_C.C_STATE > BYTE#127 THEN
		IF pi = 0 AND LOG_CL.RING_MODE THEN pi := ci; END_IF;
		pi_last := pi;
		pi := pi + 1;
		IF pi > LOG_CL.SIZE THEN pi := 1; END_IF;
		SEND := TRUE;
	ELSE
		SEND := FALSE;
	END_IF;

	TELNET_PRINT(	IP_C := IP_C,
					S_BUF := S_BUF,
					ENABLE := ENABLE,
					SEND := SEND,
					TEXT := LOG_CL.MSG[pi],
					BACK_COLOR := DWORD_TO_BYTE(SHR(LOG_CL.MSG_OPTION[pi],8)),
					FRONT_COLOR := DWORD_TO_BYTE(LOG_CL.MSG_OPTION[pi] ));
	READY := TELNET_PRINT.READY;
	done := TELNET_PRINT.DONE;

	IF SEND AND NOT done THEN
		pi := pi_last;
	END_IF;

	WATCHDOG(IN:=TRUE);

UNTIL (WATCHDOG.Q OR NOT done )
END_REPEAT;
END_FUNCTION_BLOCK

// Commented out for beedance: it uses _STRING_TO_BUFFER, which is commented out.
// FUNCTION_BLOCK TELNET_PRINT
// VAR_IN_OUT
// 	IP_C : IP_C;
// 	S_BUF : NETWORK_BUFFER;
// END_VAR
// VAR_INPUT
// 	TEXT : STRING(STRING_LENGTH);
// 	ENABLE : BOOL;
// 	SEND : BOOL;
// 	OPTION : BYTE := BYTE#2#1000_1100; (* no flush buffer (7) , CR&LF (3), Colors (2), AUTOWRAP (1), Screen-Init (0) *)
// 	BACK_COLOR : BYTE;
// 	FRONT_COLOR : BYTE;
// 	X_POS : BYTE;
// 	Y_POS : BYTE;
// 	PORT : WORD := 23; (* port number *)
// END_VAR
// VAR_OUTPUT
// 	READY : BOOL;
// 	DONE : BOOL;
// END_VAR
// VAR
// 	last_fc : BYTE;
// 	state : INT;
// 	x : INT := -1;
// 	ip_state : BYTE;
// 	ip_id : BYTE;
// 	IP_FIFO : IP_FIFO;
// 	init : BOOL;
// 	b0_screen_clear : BOOL;
// 	b1_autowrap : BOOL;
// 	b2_color : BOOL;
// 	b3_cr_lr : BOOL;
// 	b7_no_flush : BOOL;
// END_VAR
//
// READY := IP_C.C_STATE > BYTE#127;
// DONE := FALSE;
//
// CASE state OF
//
// 00: (* wait for release *)
// 	IF ENABLE THEN
// 		state := 10;
// 		ip_state := BYTE#1; (* register *)
// 	END_IF;
//
// 10: (* register with IP_Control and wait for release *)
// 	IF ip_state = BYTE#3 THEN
//
// 		(* set up IP data traffic *)
// 		IP_C.C_PORT := PORT; (* enter port number *)
// 		IP_C.C_IP := DWORD#00; (* enter IP *)
// 		IP_C.C_MODE := BYTE#4; (* Mode: TCP+PASSIV+PORT *)
// 		IP_C.TIME_RESET := TRUE; (* reset timeout monitoring *)
// 		IP_C.C_ENABLE := TRUE; (* enable connection setup *)
// 		IP_C.R_OBSERVE := FALSE; (* no receive monitoring *)
// 		state := 20;
// 	END_IF;
//
// 20:	IF IP_C.ERROR > DWORD#0 THEN
// 		IP_C.TIME_RESET := TRUE; (* reset error *)
// 	END_IF;
// 	IF S_BUF.SIZE = UINT#0 THEN (* data sending not active *)
// 		IF NOT ENABLE THEN
// 			ip_state := BYTE#4; (* close connection - release resource *)
// 			IP_C.C_ENABLE := FALSE; (* connection shutdown *)
// 			state := 0;
// 		END_IF;
// 		IF IP_C.C_STATE = BYTE#1 THEN (* rising edge connect off *)
// 			init := FALSE;
// 		ELSIF READY THEN (* connection present *)
// 			IF IP_C.C_STATE = BYTE#254 AND NOT INIT THEN (* rising edge connect on *)
// 				(* var init is necessary so the block can be called several times in the same cycle *)
// 				init := TRUE;
// 				b0_screen_clear := (OPTION AND BYTE#2#0000_0001) > BYTE#0;
// 				b1_autowrap := (OPTION AND BYTE#2#0000_0010) > BYTE#0;
// 				b2_color := (OPTION AND BYTE#2#0000_0100) > BYTE#0;
// 				b3_cr_lr := (OPTION AND BYTE#2#0000_1000) > BYTE#0;
// 				b7_no_flush := (OPTION AND BYTE#2#1000_0000) > BYTE#0;
//
// 				last_fc := NOT FRONT_COLOR; (* force color update!*)
// 				x := 0;
//
// 				(* AUTOWRAP OFF/ON *)
// 				S_BUF.BUFFER[x] := BYTE#16#1B; (* ESC *)
// 				x := x +1;
// 				S_BUF.BUFFER[x] := BYTE#16#5B; (* [ *)
// 				x := x +1;
// 				S_BUF.BUFFER[x] := BYTE#16#3F; (* ? *)
// 				x := x +1;
// 				S_BUF.BUFFER[x] := BYTE#16#37; (* 7 *)
// 				x := x +1;
// 				S_BUF.BUFFER[x] := SEL(b1_autowrap, BYTE#16#6C (* l *),BYTE#16#68 (* h *));
//
// 				IF b0_screen_clear THEN
// 					IF b2_color THEN
// 						x := x +1;
// 						S_BUF.BUFFER[x] := BYTE#16#1B; (* ESC *)
// 						x := x +1;
// 						S_BUF.BUFFER[x] := BYTE#16#5B; (* [ *)
// 						x := x +1;
// 						S_BUF.BUFFER[x] := BYTE#16#30; (* 0 *)
// 						x := x +1;
// 						S_BUF.BUFFER[x] := BYTE#16#3B; (* ; *)
// 						x := x +1;
// 						S_BUF.BUFFER[x] := BYTE#16#33; (* 3 *)
// 						x := x +1;
// 						S_BUF.BUFFER[x] := (FRONT_COLOR AND BYTE#2#00000111) OR BYTE#16#30; (* output ones digit of foreground color *)
// 						x := x +1;
// 						S_BUF.BUFFER[x] := BYTE#16#3B; (* ; *)
// 						x := x +1;
// 						S_BUF.BUFFER[x] := BYTE#16#34; (* 4 *)
// 						x := x +1;
// 						S_BUF.BUFFER[x] := (BACK_COLOR AND BYTE#2#00000111) OR BYTE#16#30; (* output ones digit of background color *)
// 						x := x +1;
// 						S_BUF.BUFFER[x] := BYTE#16#6D; (* m *)
// 					END_IF;
// 					(* Screen Clear *)
// 					x := x +1;
// 					S_BUF.BUFFER[x] := BYTE#16#1B; (* ESC *)
// 					x := x +1;
// 					S_BUF.BUFFER[x] := BYTE#16#5B; (* [ *)
// 					x := x +1;
// 					S_BUF.BUFFER[x] := BYTE#16#32; (* 2 *)
// 					x := x +1;
// 					S_BUF.BUFFER[x] := BYTE#16#4A; (* J *)
// 				ELSE
// 					x := x +1;
// 					S_BUF.BUFFER[x] := BYTE#16#0A; (* new line *)
// 				END_IF;
// 			END_IF;
//
// 			(* buffer full, or data present and no further send request *)
// 			IF (INT_TO_UINT(x + LEN(TEXT) + 21) > SIZEOF(S_BUF.BUFFER)) OR (x >= 0 AND NOT SEND) THEN
// 				S_BUF.SIZE := INT_TO_UINT(x + 1); (* enter length -> start sending data *)
// 				x := -1;
// 			ELSIF SEND THEN
//
// 				(* determine current color  *)
// 				IF b2_color AND FRONT_COLOR <> last_FC THEN
// 					(* color setting: output ANSI sequence ESC[X;Y;Zm *)
// 					x := x + 1;
// 					S_BUF.BUFFER[x] := BYTE#16#1B; (* ESC *)
// 					x := x + 1;
// 					S_BUF.BUFFER[x] := BYTE#16#5B; (* [ *)
// 					(* color setting: determine dark or bright and blinking *)
// 					IF ((FRONT_COLOR AND BYTE#2#0001_1000) XOR (last_FC AND BYTE#2#0001_1000)) <> BYTE#00 OR TRUE THEN
// 						x := x + 1;
// 						S_BUF.BUFFER[x] := BYTE#16#30; (* 0  *)
// 						x := x + 1;
// 						S_BUF.BUFFER[x] := BYTE#16#3B; (* ; *)
// 						(* no dark colors wanted -> then bold & bright *)
// 						IF (FRONT_COLOR AND BYTE#2#00001000) = BYTE#0 THEN
// 							(* switch to bold & bright colors *)
// 							x := x + 1;
// 							S_BUF.BUFFER[x] := BYTE#16#31; (* 1 *)
// 							x := x + 1;
// 							S_BUF.BUFFER[x] := BYTE#16#3B; (* ; *)
// 						END_IF;
// 						(* blinking colors wanted *)
// 						IF (FRONT_COLOR AND BYTE#2#00010000) > BYTE#0 THEN
// 							(* switch to blinking color *)
// 							x := x + 1;
// 							S_BUF.BUFFER[x] := BYTE#16#35; (* 5 *)
// 							x := x + 1;
// 							S_BUF.BUFFER[x] := BYTE#16#3B; (* ; *)
// 						END_IF;
// 					END_IF;
// 					(* output tens digit of foreground color *)
// 					x := x + 1;
// 					S_BUF.BUFFER[x] := BYTE#16#33; (* 3 *)
// 					(* output ones digit of foreground color *)
// 					x := x + 1;
// 					S_BUF.BUFFER[x] := (FRONT_COLOR AND BYTE#2#00000111) OR BYTE#16#30;
// 					x := x + 1;
// 					S_BUF.BUFFER[x] := BYTE#16#6D; (* m *)
// 					(* store new color as last used *)
// 					last_FC := FRONT_COLOR;
// 				END_IF;
//
// 				(* position cursor *)
// 				IF X_POS > BYTE#0 AND Y_POS > BYTE#0 THEN
// 					x := x + 1;
// 					S_BUF.BUFFER[x] := BYTE#16#1B; (* ESC *)
// 					x := x + 1;
// 					S_BUF.BUFFER[x] := BYTE#16#5B; (* [ *)
// 					(* output tens digit of Y_POS *)
// 					x := x + 1;
// 					S_BUF.BUFFER[x] := SHR(INT_TO_BCDC(BYTE_TO_INT(Y_POS)),4) OR BYTE#16#30;
// 					(* output ones digit of Y_POS *)
// 					x := x + 1;
// 					S_BUF.BUFFER[x] := (INT_TO_BCDC(BYTE_TO_INT(Y_POS)) AND BYTE#16#0F) OR BYTE#16#30;
// 					x := x + 1;
// 					S_BUF.BUFFER[x] := BYTE#16#3B; (* ; *)
// 					(* output tens digit of X_POS *)
// 					x := x + 1;
// 					S_BUF.BUFFER[x] := SHR(INT_TO_BCDC(BYTE_TO_INT(X_POS)),4) OR BYTE#16#30;
// 					(* output ones digit of X_POS *)
// 					x := x + 1;
// 					S_BUF.BUFFER[x] := (INT_TO_BCDC(BYTE_TO_INT(X_POS)) AND BYTE#16#0F) OR BYTE#16#30;
// 					x := x + 1;
// 					S_BUF.BUFFER[x] := BYTE#16#48; (* H *)
// 				END_IF;
//
// 				(* output text *)
// 				IF LEN(TEXT) > 0 THEN
// 					_STRING_TO_BUFFER(str:=TEXT,pos:=x + 1,pt :=REF(S_BUF.BUFFER), size:=SIZEOF(S_BUF.BUFFER));
// 					x := x + LEN(TEXT);
// 				END_IF;
//
// 				IF b3_cr_lr THEN (* Option: output CR,LF *)
// 					x := x + 1;
// 					S_BUF.BUFFER[x] := BYTE#16#0D;
// 					x := x + 1;
// 					S_BUF.BUFFER[x] := BYTE#16#0A;
// 				END_IF;
//
// 				DONE := TRUE; (* finished entering into buffer *)
//
// 				IF b7_no_flush THEN (* Option: no buffer flush *)
// 					(* send buffer immediately - store current write index -> trigger send *)
// 					S_BUF.SIZE := INT_TO_UINT(x + 1);
// 					x := -1;
// 				END_IF;
// 			END_IF;
// 		END_IF;
// 	END_IF;
// END_CASE;
//
// (* IP_FIFO *)
// IP_FIFO(FIFO:=IP_C.FIFO,STATE:=ip_state,ID:=ip_id);
// END_FUNCTION_BLOCK

// Commented out for beedance: it uses TN_INPUT_MENU_BAR, which is commented out.
// FUNCTION_BLOCK TN_FRAMEWORK
// VAR
// 	FB_IP_CONTROL : IP_CONTROL;
// 	FB_TN_INPUT_CONTROL : TN_INPUT_CONTROL;
// 	FB_TN_INPUT_MENU_BAR : TN_INPUT_MENU_BAR;
// 	FB_TN_RECEIVE :	TN_RECEIVE;
// 	FB_TN_SEND_ROWS : TN_SEND_ROWS;
// 	t : TON;
// END_VAR
// VAR_IN_OUT
// 	us_TN_INPUT_CONTROL : us_TN_INPUT_CONTROL;
// 	us_TN_SCREEN : us_TN_SCREEN;
// 	us_TN_MENU : us_TN_MENU;
// 	S_BUF : NETWORK_BUFFER;
// 	R_BUF : NETWORK_BUFFER;
// 	IP_C : IP_C;
// END_VAR
// VAR_INPUT
// 	PORT : WORD;
// END_VAR
//
// (* initialization / release of the connection *)
// IF (NOT IP_C.C_ENABLE) THEN
//
// 	(* set up IP data traffic *)
// 	IP_C.C_PORT := SEL(PORT=BYTE#0,PORT,WORD#23); (* enter port number *)
// 	IP_C.C_IP := DWORD#00; (* enter IP *)
// 	IP_C.C_MODE := BYTE#4; (* Mode: TCP+PASSIV+PORT *)
// 	IP_C.TIME_RESET := TRUE; (* reset timeout monitoring *)
// 	IP_C.C_ENABLE := TRUE; (* enable connection setup *)
// 	IP_C.R_OBSERVE := FALSE; (* no receive monitoring *)
//
// END_IF;
//
// t(IN:= IP_C.ERROR > DWORD#0, PT:=T#5s);
// IF t.Q THEN
// 	IP_C.TIME_RESET := TRUE; (* Error Reset *)
// END_IF;
//
// (* Telnet-Menu-Bar *)
// FB_TN_INPUT_MENU_BAR(
// 	Xus_TN_MENU := us_TN_MENU,
// 	Xus_TN_SCREEN := us_TN_SCREEN);
//
// (* Telnet-Input-Control *)
// FB_TN_INPUT_CONTROL(
// 	Xus_TN_SCREEN := us_TN_SCREEN,
// 	Xus_TN_INPUT_CONTROL := us_TN_INPUT_CONTROL);
//
// (* Telnet-Data-Send Line-Updates *)
// FB_TN_SEND_ROWS(
// 	IP_C :=IP_C,
// 	S_BUF :=S_BUF,
// 	Xus_TN_SCREEN :=us_TN_SCREEN,
// 	S_BUF_SIZE :=SIZEOF(S_BUF.BUFFER));
//
// (* Telnet-Server *)
// FB_IP_CONTROL(
// 	IP_C :=IP_C,
// 	S_BUF :=S_BUF,
// 	R_BUF :=R_BUF,
// 	IP :=DWORD#00,
// 	PORT :=WORD#00,
// 	TIME_OUT :=T#2s);
//
// (* Telnet-Data-Receive *)
// FB_TN_RECEIVE(
// 	R_BUF := R_BUF,
// 	Xus_TN_SCREEN := us_TN_SCREEN);
// END_FUNCTION_BLOCK

// Commented out for beedance: it uses TN_INPUT_SELECT_POPUP, which is commented out.
// FUNCTION_BLOCK TN_INPUT_CONTROL
// VAR_IN_OUT
// 	Xus_TN_SCREEN : us_TN_SCREEN;
// 	Xus_TN_INPUT_CONTROL : us_TN_INPUT_CONTROL;
// END_VAR
// VAR
// 	FB_TN_INPUT_SELECT_POPUP : TN_INPUT_SELECT_POPUP;
// 	FB_TN_INPUT_SELECT_TEXT : TN_INPUT_SELECT_TEXT;
// 	FB_TN_SC_WRITE_C : TN_SC_WRITE_C;
// 	FB_TN_INPUT_EDIT_LINE : TN_INPUT_EDIT_LINE;
// END_VAR
// VAR
// 	in_index : INT;
// 	in_Scroll_Offset : INT;
// 	in_Focus_new : INT;
// 	in_Focus_alt : INT;
// 	bo_Tool_Tip_Update : BOOL;
// END_VAR
//
// (* processing enabled? *)
// IF (Xus_TN_INPUT_CONTROL.bo_Enable = FALSE) OR (Xus_TN_SCREEN.bo_Menue_Bar_Dialog = TRUE) THEN
// 	RETURN;
// END_IF;
//
// (* perform focus reset *)
// IF (Xus_TN_INPUT_CONTROL.bo_Reset_Fokus = TRUE) THEN
// 	Xus_TN_INPUT_CONTROL.bo_Reset_Fokus := FALSE;
//
// 	FOR in_index := INT#01 TO Xus_TN_INPUT_CONTROL.in_Count DO
// 		Xus_TN_INPUT_CONTROL.usa_TN_INPUT_CONTROL_DATA[in_index].bo_Focus := FALSE;
// 	END_FOR;
//
// 	IF (Xus_TN_INPUT_CONTROL.in_Count >= INT#01) THEN
// 		Xus_TN_INPUT_CONTROL.usa_TN_INPUT_CONTROL_DATA[1].bo_Focus := TRUE;
// 		Xus_TN_INPUT_CONTROL.in_Focus_at := INT#01;
// 	END_IF;
//
// 	Xus_TN_INPUT_CONTROL.bo_Update_all := TRUE;
// END_IF;
//
// IF (Xus_TN_SCREEN.bo_Modal_Dialog = FALSE) THEN
// 	(* evaluate TAB key for switching control element *)
// 	IF (Xus_TN_SCREEN.by_Input_Exten_Code = BYTE#09) THEN
//
// 		in_Scroll_Offset := INT#01;
//
// 		(* cursor up key *)
// 	ELSIF (Xus_TN_SCREEN.by_Input_Exten_Code = BYTE#65) THEN
//
// 		in_Scroll_Offset := -1;
//
// 		(* cursor down key *)
// 	ELSIF (Xus_TN_SCREEN.by_Input_Exten_Code = BYTE#66) THEN
//
// 		in_Scroll_Offset := INT#01;
//
// 	END_IF;
// END_IF;
//
// IF (in_Scroll_Offset <> INT#00) THEN
// 	(* check limits                                            *)
//
// 	Xus_TN_INPUT_CONTROL.in_Focus_at:=LIMIT(INT#01,Xus_TN_INPUT_CONTROL.in_Focus_at,Xus_TN_INPUT_CONTROL.in_Count);
//
// 	in_Focus_new := Xus_TN_INPUT_CONTROL.in_Focus_at + in_Scroll_Offset;
//
// 	IF (in_Focus_new > Xus_TN_INPUT_CONTROL.in_Count) THEN
// 		in_Focus_new := INT#1;
// 	END_IF;
//
// 	IF (in_Focus_new < INT#01) THEN
// 		in_Focus_new := Xus_TN_INPUT_CONTROL.in_Count;
// 	END_IF;
//
// 	in_Focus_alt := Xus_TN_INPUT_CONTROL.in_Focus_at;
//
// 	(* remove focus from the current element *)
// 	Xus_TN_INPUT_CONTROL.usa_TN_INPUT_CONTROL_DATA[in_Focus_alt].bo_Focus := FALSE;
// 	Xus_TN_INPUT_CONTROL.usa_TN_INPUT_CONTROL_DATA[in_Focus_alt].bo_Update_Input := TRUE;
//
// 	(* give focus to the new element *)
// 	Xus_TN_INPUT_CONTROL.usa_TN_INPUT_CONTROL_DATA[in_Focus_new].bo_Focus  := TRUE;
// 	Xus_TN_INPUT_CONTROL.usa_TN_INPUT_CONTROL_DATA[in_Focus_new].bo_Update_Input := TRUE;
//
// 	Xus_TN_INPUT_CONTROL.in_Focus_at := in_Focus_new;
//
// 	bo_Tool_Tip_Update := TRUE;
// 	in_Scroll_Offset := INT#00;
//
// END_IF;
//
// (* update all elements? *)
// IF (Xus_TN_INPUT_CONTROL.bo_Update_all = TRUE) THEN
// 	FOR in_index := 1 TO Xus_TN_INPUT_CONTROL.in_Count DO
// 		Xus_TN_INPUT_CONTROL.usa_TN_INPUT_CONTROL_DATA[in_index].bo_Update_All := TRUE;
// 	END_FOR;
// 	Xus_TN_INPUT_CONTROL.bo_Update_all := FALSE;
// 	bo_Tool_Tip_Update := TRUE;
// END_IF;
//
// FOR in_index := 1 TO Xus_TN_INPUT_CONTROL.in_Count DO
//
// 	IF (Xus_TN_INPUT_CONTROL.usa_TN_INPUT_CONTROL_DATA[in_index].in_Type > INT#00) THEN
//
// 		IF (Xus_TN_INPUT_CONTROL.usa_TN_INPUT_CONTROL_DATA[in_index].bo_Focus = TRUE) THEN
//
// 			Xus_TN_INPUT_CONTROL.usa_TN_INPUT_CONTROL_DATA[in_index].by_Input_ASCII_Code  := Xus_TN_SCREEN.by_Input_ASCII_Code;
// 			Xus_TN_INPUT_CONTROL.usa_TN_INPUT_CONTROL_DATA[in_index].by_Input_Exten_Code  := Xus_TN_SCREEN.by_Input_Exten_Code;
// 			Xus_TN_INPUT_CONTROL.usa_TN_INPUT_CONTROL_DATA[in_index].bo_Input_ASCII_IsNum := Xus_TN_SCREEN.bo_Input_ASCII_IsNum;
//
// 			(* output tooltip text *)
// 			IF (bo_Tool_Tip_Update = TRUE) THEN
//
// 				FB_TN_SC_WRITE_C(	Iin_Y := Xus_TN_INPUT_CONTROL.in_ToolTip_Y,
// 									Iin_X := Xus_TN_INPUT_CONTROL.in_ToolTip_X,
// 									Iby_ATTR := Xus_TN_INPUT_CONTROL.by_ToolTip_Attr,
// 									Iin_OPTION := INT#02, (* Center-String *)
// 									Iin_LENGTH := Xus_TN_INPUT_CONTROL.in_ToolTip_Size,
// 									Ist_STRING := Xus_TN_INPUT_CONTROL.usa_TN_INPUT_CONTROL_DATA[in_index].st_Input_ToolTip,
// 									Xus_TN_SCREEN := Xus_TN_SCREEN);
//
// 				(* reset flag *)
// 				bo_Tool_Tip_Update := FALSE;
// 			END_IF;
// 		END_IF;
//
// 		CASE Xus_TN_INPUT_CONTROL.usa_TN_INPUT_CONTROL_DATA[in_index].in_Type OF
// 		1:
// 			(* process edit line *)
// 			FB_TN_INPUT_EDIT_LINE(	Xus_TN_INPUT_CONTROL_DATA := Xus_TN_INPUT_CONTROL.usa_TN_INPUT_CONTROL_DATA[in_index],
// 									Xus_TN_SCREEN := Xus_TN_SCREEN);
// 		2:
// 			(* process select text *)
// 			FB_TN_INPUT_SELECT_TEXT(	Xus_TN_INPUT_CONTROL_DATA := Xus_TN_INPUT_CONTROL.usa_TN_INPUT_CONTROL_DATA[in_index],
// 										Xus_TN_SCREEN := Xus_TN_SCREEN);
// 		3:
// 			(* process select popup *)
// 			FB_TN_INPUT_SELECT_POPUP(	Xus_TN_INPUT_CONTROL_DATA := Xus_TN_INPUT_CONTROL.usa_TN_INPUT_CONTROL_DATA[in_index],
// 										Xus_TN_SCREEN := Xus_TN_SCREEN);
// 		END_CASE;
//
// 		IF (Xus_TN_INPUT_CONTROL.usa_TN_INPUT_CONTROL_DATA[in_index].bo_Focus = TRUE) THEN
//
// 			(* transfer cursor position of element to screen *)
// 			Xus_TN_SCREEN.in_Cursor_X := Xus_TN_INPUT_CONTROL.usa_TN_INPUT_CONTROL_DATA[in_index].in_Cursor_X;
// 			Xus_TN_SCREEN.in_Cursor_Y := Xus_TN_INPUT_CONTROL.usa_TN_INPUT_CONTROL_DATA[in_index].in_Cursor_Y;
//
// 		END_IF;
// 	END_IF;
// END_FOR;
// END_FUNCTION_BLOCK

// Commented out for beedance: it uses CHR_TO_STRING, which is commented out.
// FUNCTION_BLOCK TN_INPUT_EDIT_LINE
// VAR
// 	in_count : INT;
// 	in_Count_End : INT;
// 	in_CursorOffset : INT;
// 	by_Attr : BYTE;
// 	st_String : STRING;
// 	bo_Pos_Found : BOOL;
// 	st_CHAR : STRING(1);
// 	in_old_charpos : INT;
// END_VAR
// VAR
// 	FB_TN_SC_WRITE : TN_SC_WRITE;
// END_VAR
// VAR_IN_OUT
// 	Xus_TN_SCREEN : us_TN_SCREEN;
// 	Xus_TN_INPUT_CONTROL_DATA : us_TN_INPUT_CONTROL_DATA;
// END_VAR
//
// (* reset cursor control *)
// in_CursorOffset := INT#0;
//
// IF Xus_TN_INPUT_CONTROL_DATA.bo_Focus = TRUE THEN
//
// 	(* text input detected? *)
// 	IF Xus_TN_INPUT_CONTROL_DATA.by_Input_ASCII_Code > BYTE#0 THEN
//
// 		IF (Xus_TN_INPUT_CONTROL_DATA.bo_Input_Only_Num = TRUE AND Xus_TN_INPUT_CONTROL_DATA.bo_Input_ASCII_IsNum = TRUE)
// 			OR (Xus_TN_INPUT_CONTROL_DATA.bo_Input_Only_Num = FALSE) THEN
//
// 			(* convert ASCII value into a string *)
// 			st_CHAR := CHR_TO_STRING(C:=Xus_TN_INPUT_CONTROL_DATA.by_Input_ASCII_Code);
//
// 			(* accept input *)
// 			Xus_TN_INPUT_CONTROL_DATA.st_Input_Data := REPLACE(Xus_TN_INPUT_CONTROL_DATA.st_Input_Data,
// 			st_CHAR,INT#1,Xus_TN_INPUT_CONTROL_DATA.in_Cursor_Pos);
//
// 			in_CursorOffset := INT#1;
// 			Xus_TN_INPUT_CONTROL_DATA.bo_Update_Input := TRUE;
// 		END_IF;
// 	END_IF;
//
// 	CASE BYTE_TO_INT(Xus_TN_INPUT_CONTROL_DATA.by_Input_Exten_Code) OF
//
// 	67: (* cursor right pressed *)
// 		in_CursorOffset := INT#1;
//
// 	68: (* cursor left pressed *)
// 		in_CursorOffset := -1;
//
// 	08: (* backspace pressed *)
// 		Xus_TN_INPUT_CONTROL_DATA.st_Input_Data := REPLACE(Xus_TN_INPUT_CONTROL_DATA.st_Input_Data, ' ', 1,Xus_TN_INPUT_CONTROL_DATA.in_Cursor_Pos);
// 		Xus_TN_INPUT_CONTROL_DATA.bo_Update_Input := TRUE;
// 		in_CursorOffset := -1;
//
// 	13: (* enter key pressed *)
// 		IF LEN(Xus_TN_INPUT_CONTROL_DATA.st_Input_Mask) > INT#00 THEN
// 			(* accept input string *)
// 			Xus_TN_INPUT_CONTROL_DATA.st_Input_String := Xus_TN_INPUT_CONTROL_DATA.st_Input_Data;
//
// 			(* input string -> remove leading and trailing spaces *)
// 			Xus_TN_INPUT_CONTROL_DATA.st_Input_String := TRIME(str:=Xus_TN_INPUT_CONTROL_DATA.st_Input_String);
// 			Xus_TN_INPUT_CONTROL_DATA.bo_Input_Entered := TRUE;
//
// 			(* prepare new input *)
// 			Xus_TN_INPUT_CONTROL_DATA.st_Input_Data := Xus_TN_INPUT_CONTROL_DATA.st_Input_Mask;
//
// 			Xus_TN_INPUT_CONTROL_DATA.in_Cursor_Pos := INT#1;
// 			Xus_TN_INPUT_CONTROL_DATA.bo_Update_Input := TRUE;
//
// 			(* search first position in input mask *)
// 			st_CHAR := MID(Xus_TN_INPUT_CONTROL_DATA.st_Input_Mask,1,Xus_TN_INPUT_CONTROL_DATA.in_Cursor_Pos);
// 			IF st_CHAR <> ' ' THEN
// 				(* search next input position *)
// 				in_CursorOffset := INT#1;
// 			END_IF;
// 		END_IF;
// 	END_CASE;
// END_IF;
//
// (* move cursor to the right                                   *)
// IF (in_CursorOffset > INT#0) OR (Xus_TN_INPUT_CONTROL_DATA.in_Cursor_Pos = INT#0) THEN
// 	bo_Pos_Found := FALSE;
//
// 	in_Count := Xus_TN_INPUT_CONTROL_DATA.in_Cursor_Pos + INT#1;
// 	in_Count_End := LEN(Xus_TN_INPUT_CONTROL_DATA.st_Input_Mask);
//
// 	WHILE (in_count <= in_Count_End) AND (bo_Pos_Found = FALSE) DO
//
// 		st_CHAR := MID(Xus_TN_INPUT_CONTROL_DATA.st_Input_Mask,1,in_count);
// 		IF st_CHAR = ' ' THEN
// 			Xus_TN_INPUT_CONTROL_DATA.in_Cursor_Pos := in_count;
// 			Xus_TN_INPUT_CONTROL_DATA.bo_Update_Input := TRUE;
// 			bo_Pos_Found := TRUE;
// 		END_IF;
//
// 		in_count := in_count + INT#1;
//
// 	END_WHILE;
// END_IF;
//
// (* move cursor to the left *)
// IF in_CursorOffset < INT#0 THEN
// 	bo_Pos_Found := FALSE;
//
// 	in_Count     := Xus_TN_INPUT_CONTROL_DATA.in_Cursor_Pos - INT#01;
// 	in_Count_End := INT#1;
//
// 	WHILE (in_count >= in_Count_End) AND (bo_Pos_Found = FALSE) DO
//
// 		st_CHAR := MID(Xus_TN_INPUT_CONTROL_DATA.st_Input_Mask,1,in_count);
// 		IF st_CHAR = ' ' THEN
// 			Xus_TN_INPUT_CONTROL_DATA.in_Cursor_Pos := in_count;
// 			Xus_TN_INPUT_CONTROL_DATA.bo_Update_Input := TRUE;
// 			bo_Pos_Found := TRUE;
// 		END_IF;
//
// 		in_count := in_count - INT#1;
// 	END_WHILE;
// END_IF;
//
// (* maximum cursor position? *)
// IF Xus_TN_INPUT_CONTROL_DATA.in_Cursor_Pos > LEN(Xus_TN_INPUT_CONTROL_DATA.st_Input_Data) THEN
// 	Xus_TN_INPUT_CONTROL_DATA.in_Cursor_Pos := LEN(Xus_TN_INPUT_CONTROL_DATA.st_Input_Data);
// 	Xus_TN_INPUT_CONTROL_DATA.bo_Update_Input := TRUE;
// END_IF;
//
// (* minimum cursor position? *)
// IF Xus_TN_INPUT_CONTROL_DATA.in_Cursor_Pos < INT#1 THEN
// 	Xus_TN_INPUT_CONTROL_DATA.in_Cursor_Pos := INT#1;
// 	Xus_TN_INPUT_CONTROL_DATA.bo_Update_Input := TRUE;
// END_IF;
//
// (* update of the display *)
// IF (Xus_TN_INPUT_CONTROL_DATA.bo_Update_Input = TRUE) OR (Xus_TN_INPUT_CONTROL_DATA.bo_Update_All = TRUE) THEN
//
// 	(* output title text *)
// 	IF (Xus_TN_INPUT_CONTROL_DATA.bo_Update_All = TRUE) THEN
//
// 		IF (Xus_TN_INPUT_CONTROL_DATA.in_Title_X_Offset = INT#00) AND (Xus_TN_INPUT_CONTROL_DATA.in_Title_Y_Offset = INT#00) THEN
// 			(* if offset X,Y = 0 then position the title string left of the element *)
// 			FB_TN_SC_WRITE.Iin_Y := Xus_TN_INPUT_CONTROL_DATA.in_Y;
// 			FB_TN_SC_WRITE.Iin_X := Xus_TN_INPUT_CONTROL_DATA.in_X - LEN(Xus_TN_INPUT_CONTROL_DATA.st_Title_String);
// 		ELSE
// 			(* output title text via row, color offset *)
// 			FB_TN_SC_WRITE.Iin_Y := Xus_TN_INPUT_CONTROL_DATA.in_Y + Xus_TN_INPUT_CONTROL_DATA.in_Title_Y_Offset;
// 			FB_TN_SC_WRITE.Iin_X := Xus_TN_INPUT_CONTROL_DATA.in_X + Xus_TN_INPUT_CONTROL_DATA.in_Title_X_Offset;
// 		END_IF;
//
// 		(* output title text via row, color offset *)
// 		FB_TN_SC_WRITE(	Iby_ATTR := Xus_TN_INPUT_CONTROL_DATA.by_Title_Attr,
// 						Ist_STRING := Xus_TN_INPUT_CONTROL_DATA.st_Title_String,
// 						Xus_TN_SCREEN := Xus_TN_SCREEN);
// 	END_IF;
//
// 	(* output input text *)
// 	IF (Xus_TN_INPUT_CONTROL_DATA.bo_Input_Hidden = TRUE) THEN
//
// 		st_String := '';
//
// 		IF LEN(Xus_TN_INPUT_CONTROL_DATA.st_Input_Data) = LEN(Xus_TN_INPUT_CONTROL_DATA.st_Input_Mask) THEN
// 			(* input mode: HIDDEN *)
// 			FOR in_count := 1 TO LEN(Xus_TN_INPUT_CONTROL_DATA.st_Input_Data) DO
//
// 				(* read character from input mask *)
// 				st_CHAR := MID(Xus_TN_INPUT_CONTROL_DATA.st_Input_Mask,1,in_count);
//
// 				(* output input or mask character *)
// 				IF st_CHAR = ' ' THEN
//
// 					(* read character from input data *)
// 					st_CHAR := MID(Xus_TN_INPUT_CONTROL_DATA.st_Input_Data,1,in_count);
//
// 					IF st_CHAR = ' ' THEN
// 						(* output spaces *)
// 						st_String := CONCAT(st_String, ' ');
//
// 					ELSE
// 						(* output hidden character *)
// 						st_String := CONCAT(st_String, '*');
//
// 					END_IF;
//
// 				ELSE
// 					(* take character from input mask *)
// 					st_CHAR := MID(Xus_TN_INPUT_CONTROL_DATA.st_Input_Data,1,in_count);
// 					st_String := CONCAT(st_String,st_CHAR);
//
// 				END_IF;
// 			END_FOR;
// 		END_IF;
// 	ELSE
//
// 		(* input mode: NORMAL *)
// 		st_String := Xus_TN_INPUT_CONTROL_DATA.st_Input_Data;
//
// 	END_IF;
//
// 	(* output string *)
//
// 	IF Xus_TN_INPUT_CONTROL_DATA.bo_Focus = TRUE THEN
// 		by_Attr := Xus_TN_INPUT_CONTROL_DATA.by_Attr_mF;
// 	ELSE
// 		by_Attr := Xus_TN_INPUT_CONTROL_DATA.by_Attr_oF;
// 	END_IF;
//
// 	FB_TN_SC_WRITE(	Iin_Y := Xus_TN_INPUT_CONTROL_DATA.in_Y,
// 					Iin_X := Xus_TN_INPUT_CONTROL_DATA.in_X,
// 					Iby_ATTR := by_Attr,
// 					Ist_STRING := st_String,
// 					Xus_TN_SCREEN := Xus_TN_SCREEN);
//
// 	(* set cursor to current position *)
// 	Xus_TN_INPUT_CONTROL_DATA.in_Cursor_Y := Xus_TN_INPUT_CONTROL_DATA.in_Y;
// 	Xus_TN_INPUT_CONTROL_DATA.in_Cursor_X := Xus_TN_INPUT_CONTROL_DATA.in_X + Xus_TN_INPUT_CONTROL_DATA.in_Cursor_Pos - INT#1;
//
// 	in_old_charpos := INT#0;
//
// 	(* reset update flags *)
// 	Xus_TN_INPUT_CONTROL_DATA.bo_Update_All := FALSE;
// 	Xus_TN_INPUT_CONTROL_DATA.bo_Update_Input := FALSE;
// END_IF;
// END_FUNCTION_BLOCK

// Commented out for beedance: it uses ELEMENT_GET, which is commented out.
// FUNCTION_BLOCK TN_INPUT_MENU_BAR
// VAR
// 	FB_TN_INPUT_MENU_POPUP : TN_INPUT_MENU_POPUP;
// 	us_TN_MENU_POPUP : us_TN_MENU_POPUP;
// 	FB_TN_SC_WRITE_C : TN_SC_WRITE_C;
// END_VAR
// VAR
// 	in_ROW : INT;
// 	in_COL : INT;
// 	in_TITLE_Length : INT;
// 	st_MENU_BAR : STRING(STRING_LENGTH);
// 	st_MENU_TITLE : STRING;
// 	in_Count : INT;
// 	in_Index : INT;
// 	by_New_KeyCode : BYTE;
// 	in_Scroll_Offset : INT;
// 	by_ATTR : BYTE;
// 	bo_Reset_Position :	BOOL;
// END_VAR
// VAR_IN_OUT
// 	Xus_TN_MENU : us_TN_MENU;
// 	Xus_TN_SCREEN : us_TN_SCREEN;
// END_VAR
//
// (* make sure the rectangle is always positioned inside the screen *)
//
// IF (Xus_TN_MENU.in_State = INT#00) AND (Xus_TN_MENU.bo_Create = TRUE) THEN
// 	Xus_TN_MENU.in_State := INT#01;
// 	Xus_TN_MENU.bo_Create := FALSE;
// 	Xus_TN_MENU.in_Menu_Selected := INT#00;
// 	Xus_TN_MENU.bo_Update := TRUE;
// 	bo_Reset_Position := TRUE;
//
// 	(* menu bar - main menu *)
// 	st_MENU_BAR := ELEMENT_GET(SEP:=BYTE#37,POS:=0,ELEMENT:=Xus_TN_MENU.st_MENU_TEXT);
//
// 	(* menu bar - determine number of elements *)
// 	Xus_TN_MENU.in_Menu_E_Count := ELEMENT_COUNT(SEP:=BYTE#35,ELEMENT:=st_MENU_BAR);
//
// END_IF;
//
// (* store keycode *)
// by_New_KeyCode := Xus_TN_SCREEN.by_Input_Exten_Code;
//
// (* popup menu key control (only allow cursor up + down *)
// IF (by_New_KeyCode = BYTE#65) OR (by_New_KeyCode = BYTE#66) THEN
// 	us_TN_MENU_POPUP.by_Input_Exten_Code := by_New_KeyCode;
// ELSE
// 	us_TN_MENU_POPUP.by_Input_Exten_Code := BYTE#00;
// END_IF;
//
// (* Escape *)
// IF (by_New_KeyCode = BYTE#27) THEN
// 	(* menu was inactive -> escape -> activate menu *)
// 	IF (Xus_TN_MENU.in_State = INT#01) AND (Xus_TN_SCREEN.bo_Modal_Dialog = FALSE) THEN
// 		Xus_TN_MENU.in_State := INT#02;
// 		Xus_TN_MENU.bo_Update := TRUE;
// 		Xus_TN_MENU.in_Menu_Selected := INT#00;
//
// 		Xus_TN_SCREEN.bo_Menue_Bar_Dialog := TRUE;
//
// 		(* menu was active -> escape -> deactivate menu *)
// 	ELSIF (Xus_TN_MENU.in_State = INT#02) THEN
// 		us_TN_MENU_POPUP.bo_Destroy := TRUE;
// 		Xus_TN_MENU.bo_Update := TRUE;
// 		Xus_TN_MENU.in_State := INT#01;
// 		bo_Reset_Position := TRUE;
//
// 		Xus_TN_SCREEN.bo_Menue_Bar_Dialog := FALSE;
// 	END_IF;
// END_IF;
//
// (* menu active *)
// IF (Xus_TN_MENU.in_State = INT#02) THEN
//
// 	(* Return *)
// 	IF (by_New_KeyCode = BYTE#13)  THEN
// 		us_TN_MENU_POPUP.bo_Destroy := TRUE;
// 		Xus_TN_MENU.bo_Update := TRUE;
// 		Xus_TN_MENU.in_State := INT#01;
// 		bo_Reset_Position := TRUE;
// 		Xus_TN_MENU.in_Menu_Selected := (Xus_TN_MENU.in_Cur_Menu_Item * INT#10) + Xus_TN_MENU.in_Cur_Sub_Item;
// 		Xus_TN_SCREEN.by_Input_Exten_Code := BYTE#00;
//
// 		Xus_TN_SCREEN.bo_Menue_Bar_Dialog := FALSE;
//
// 		(* destroy command -> close popup menu *)
// 	ELSIF (Xus_TN_MENU.bo_Destroy = TRUE) THEN
// 		us_TN_MENU_POPUP.bo_Destroy := TRUE;
// 		Xus_TN_MENU.bo_Update := TRUE;
// 		Xus_TN_MENU.in_State := INT#01;
// 		bo_Reset_Position := TRUE;
// 		Xus_TN_MENU.in_Menu_Selected := INT#00;
// 		Xus_TN_SCREEN.by_Input_Exten_Code := BYTE#00;
//
// 		Xus_TN_SCREEN.bo_Menue_Bar_Dialog := FALSE;
//
// 	END_IF;
//
// 	IF (by_New_KeyCode = BYTE#67) THEN (* cursor right *)
// 		in_Scroll_Offset := INT#1;
// 		Xus_TN_MENU.bo_Update := TRUE;
// 		Xus_TN_SCREEN.by_Input_Exten_Code := BYTE#00;
//
// 	ELSIF (by_New_KeyCode = BYTE#68) THEN (* cursor left *)
// 		in_Scroll_Offset := -1;
// 		Xus_TN_MENU.bo_Update := TRUE;
// 		Xus_TN_SCREEN.by_Input_Exten_Code := BYTE#00;
// 	END_IF;
// END_IF;
//
// IF bo_Reset_Position = TRUE THEN
// 	bo_Reset_Position := FALSE;
// 	Xus_TN_MENU.in_X_SM_old := -1;
// 	Xus_TN_MENU.in_Y_SM_old := -1;
// 	Xus_TN_MENU.in_X_SM_new := -1;
// 	Xus_TN_MENU.in_Y_SM_new := -1;
// END_IF;
//
// (* update POPUP menu *)
// IF (Xus_TN_MENU.in_State > INT#00) AND (Xus_TN_MENU.bo_Update = TRUE) THEN
//
// 	Xus_TN_MENU.bo_Update := FALSE;
//
// 	in_ROW := Xus_TN_MENU.in_Y;
// 	in_COL := Xus_TN_MENU.in_X;
//
// 	(* Scrolloffset *)
// 	IF in_Scroll_Offset <> INT#00 THEN
// 		Xus_TN_MENU.in_Cur_Menu_Item := INC2(Xus_TN_MENU.in_Cur_Menu_Item,in_Scroll_Offset,1,Xus_TN_MENU.in_Menu_E_Count);
// 		in_Scroll_Offset := INT#00;
// 	ELSE
// 		(* item = 0 and no scroll offset *)
// 		IF (Xus_TN_MENU.in_Cur_Menu_Item = INT#00) THEN
// 			Xus_TN_MENU.in_Cur_Menu_Item := INT#01;
// 		END_IF;
// 	END_IF;
//
// 	(* draw all menu texts *)
// 	FOR in_Count := INT#01 TO Xus_TN_MENU.in_Menu_E_Count DO;
//
// 		(* determine character color *)
// 		IF (in_Count = Xus_TN_MENU.in_Cur_Menu_Item) AND (Xus_TN_MENU.in_State > INT#01 ) THEN
// 			by_ATTR := Xus_TN_MENU.by_Attr_mF;
//
// 			Xus_TN_MENU.in_Y_SM_new := in_ROW + INT#01;
// 			Xus_TN_MENU.in_X_SM_new := in_COL;
//
// 		ELSE
// 			by_ATTR := Xus_TN_MENU.by_Attr_oF;
// 		END_IF;
//
// 		st_MENU_TITLE := ELEMENT_GET(SEP:=BYTE#35,POS:=in_Count - 1,ELEMENT:=st_MENU_BAR);
//
// 		in_TITLE_Length := LEN(st_MENU_TITLE) + INT#02;
//
// 		FB_TN_SC_WRITE_C(	Iin_Y := in_ROW,
// 							Iin_X := in_COL,
// 							Iby_ATTR := by_ATTR,
// 							Iin_LENGTH := in_TITLE_Length,
// 							Iin_OPTION := INT#02,
// 							Ist_STRING := st_MENU_TITLE,
// 							Xus_TN_SCREEN := Xus_TN_SCREEN);
//
// 		in_COL := in_COL + in_TITLE_Length;
//
// 	END_FOR;
// END_IF;
//
// IF Xus_TN_MENU.in_X_SM_new <> Xus_TN_MENU.in_X_SM_old THEN
//
// 	(* submenu is active -> exit                                     *)
// 	IF us_TN_MENU_POPUP.bo_Activ = TRUE THEN
// 		us_TN_MENU_POPUP.bo_Destroy := TRUE;
//
// 		(* process submenu *)
// 		FB_TN_INPUT_MENU_POPUP(	Xus_TN_MENU_POPUP := us_TN_MENU_POPUP,
// 								Xus_TN_SCREEN := Xus_TN_SCREEN);
// 	END_IF;
//
// 	IF us_TN_MENU_POPUP.bo_Activ = FALSE THEN
// 		(* configure and run the popup menu for the current menu         *)
// 		in_Index := Xus_TN_MENU.in_Cur_Menu_Item;
//
// 		us_TN_MENU_POPUP.in_Y := Xus_TN_MENU.in_Y_SM_new;
// 		us_TN_MENU_POPUP.in_X := Xus_TN_MENU.in_X_SM_new;
// 		us_TN_MENU_POPUP.by_Attr_mF := Xus_TN_MENU.by_Attr_mF;
// 		us_TN_MENU_POPUP.by_Attr_oF := Xus_TN_MENU.by_Attr_oF;
// 		us_TN_MENU_POPUP.st_Menu_Text := ELEMENT_GET(SEP:=BYTE#37,POS:=in_Index,ELEMENT:=Xus_TN_MENU.st_MENU_TEXT);
// 		us_TN_MENU_POPUP.bo_Create := TRUE;
//
// 		Xus_TN_MENU.in_X_SM_old := Xus_TN_MENU.in_X_SM_new;
// 		Xus_TN_MENU.in_Y_SM_old := Xus_TN_MENU.in_Y_SM_new;
//
// 	END_IF;
// END_IF;
//
// (* call popup menu cyclically *)
// FB_TN_INPUT_MENU_POPUP(	Xus_TN_MENU_POPUP := us_TN_MENU_POPUP,
// 						Xus_TN_SCREEN := Xus_TN_SCREEN);
//
// (* copy current item from popup menu *)
// Xus_TN_MENU.in_Cur_Sub_Item := us_TN_MENU_POPUP.in_Cur_Item;
//
// (* destroy command *)
// IF (Xus_TN_MENU.in_State = INT#01) THEN
// 	IF (Xus_TN_MENU.bo_Destroy = TRUE) THEN
// 		Xus_TN_MENU.in_State := INT#00;
// 		Xus_TN_MENU.bo_Destroy := FALSE;
// 		Xus_TN_MENU.in_Cur_Menu_Item := INT#00;
// 		Xus_TN_MENU.in_Cur_Sub_Item := INT#00;
// 	END_IF;
// END_IF;
// END_FUNCTION_BLOCK

// Commented out for beedance: it uses ELEMENT_COUNT, which is commented out.
// FUNCTION_BLOCK TN_INPUT_MENU_POPUP
// VAR
// 	FB_TN_SC_AREA_SAVE : TN_SC_AREA_SAVE;
// 	FB_TN_SC_AREA_RESTORE : TN_SC_AREA_RESTORE;
// 	FB_TN_SC_LINE : TN_SC_LINE;
// 	FB_TN_SC_ADD_SHADOW : TN_SC_ADD_SHADOW;
// 	FB_TN_SC_BOX : TN_SC_BOX;
// 	FB_TN_SC_WRITE_C : TN_SC_WRITE_C;
// END_VAR
// VAR
// 	in_ROW : INT;
// 	in_ROWS : INT;
// 	in_COL : INT;
// 	in_COLS : INT;
// 	in_index : INT;
// 	in_Count : INT;
// 	in_Scroll_Offset : INT;
// 	by_ATTR : BYTE;
// END_VAR
// VAR_IN_OUT
// 	Xus_TN_MENU_POPUP : us_TN_MENU_POPUP;
// 	Xus_TN_SCREEN : us_TN_SCREEN;
// END_VAR
//
// (* make sure the rectangle is always positioned inside the screen *)
//
// IF (Xus_TN_MENU_POPUP.bo_Activ = FALSE) AND (Xus_TN_MENU_POPUP.bo_Create = TRUE) THEN
// 	Xus_TN_MENU_POPUP.bo_Activ := TRUE;
// 	Xus_TN_MENU_POPUP.bo_Create := FALSE;
// 	Xus_TN_MENU_POPUP.bo_Destroy := FALSE;
// 	Xus_TN_MENU_POPUP.bo_Update := TRUE;
//
//   (* submenu texts *)
//
// 	Xus_TN_MENU_POPUP.in_Menu_E_Count := ELEMENT_COUNT(SEP:=BYTE#35,ELEMENT:=Xus_TN_MENU_POPUP.st_Menu_Text);
//
// 	(* determine number of lines (submenu texts) *)
// 	Xus_TN_MENU_POPUP.in_Rows := Xus_TN_MENU_POPUP.in_Menu_E_Count;
//
// 	(* find longest submenu text *)
// 	Xus_TN_MENU_POPUP.in_Cols := INT#00;
//
// 	FOR in_Count := INT#01 TO Xus_TN_MENU_POPUP.in_Rows DO;
// 		Xus_TN_MENU_POPUP.in_Cols:=MAX(LEN(ELEMENT_GET(SEP:=BYTE#35,POS:=in_Count - 1,ELEMENT:=Xus_TN_MENU_POPUP.st_Menu_Text)),Xus_TN_MENU_POPUP.in_Cols);
// 	END_FOR;
//
// 	(* check and correct horizontal position *)
// 	IF (Xus_TN_MENU_POPUP.in_X + Xus_TN_MENU_POPUP.in_Cols) > INT#75 THEN
// 		Xus_TN_MENU_POPUP.in_X := INT#79 - Xus_TN_MENU_POPUP.in_Cols - INT#04;
// 	END_IF;
//
//   (* check and correct vertical position *)
// 	IF (Xus_TN_MENU_POPUP.in_Y + Xus_TN_MENU_POPUP.in_ROWS) > INT#21 THEN
// 		Xus_TN_MENU_POPUP.in_Y := INT#23 - Xus_TN_MENU_POPUP.in_ROWS - INT#2;
// 	END_IF;
//
// 	Xus_TN_SCREEN.bo_Modal_Dialog := TRUE;
//
// 	(* save background *)
// 	FB_TN_SC_AREA_SAVE(	Iin_X1 := Xus_TN_MENU_POPUP.in_X,
// 									Iin_Y1 := Xus_TN_MENU_POPUP.in_Y,
// 									Iin_X2 := Xus_TN_MENU_POPUP.in_X + Xus_TN_MENU_POPUP.in_Cols + INT#04,
// 									Iin_Y2 := Xus_TN_MENU_POPUP.in_Y + Xus_TN_MENU_POPUP.in_Rows + INT#02,
// 									Xus_TN_SCREEN := Xus_TN_SCREEN);
//
// 	(* draw frame for submenu *)
// 	FB_TN_SC_BOX(	Iin_X1 := Xus_TN_MENU_POPUP.in_X,
// 					Iin_Y1 := Xus_TN_MENU_POPUP.in_Y,
// 					Iin_X2 := Xus_TN_MENU_POPUP.in_X + Xus_TN_MENU_POPUP.in_Cols + INT#03,
// 					Iin_Y2 := Xus_TN_MENU_POPUP.in_Y + Xus_TN_MENU_POPUP.in_Rows + INT#01,
// 					Iby_FILL := BYTE#32, (* fill *)
// 					Iin_BORDER := INT#01, (* Single-Line Border *)
// 					Iby_ATTR := Xus_TN_MENU_POPUP.by_Attr_oF,
// 					Xus_TN_SCREEN := Xus_TN_SCREEN);
//
// 	(* draw shadow for submenu *)
// 	FB_TN_SC_ADD_SHADOW(Iin_X1 := Xus_TN_MENU_POPUP.in_X + INT#1,
// 						Iin_Y1 := Xus_TN_MENU_POPUP.in_Y + INT#1,
// 						Iin_X2 := Xus_TN_MENU_POPUP.in_X + Xus_TN_MENU_POPUP.in_Cols + INT#04,
// 						Iin_Y2 := Xus_TN_MENU_POPUP.in_Y + Xus_TN_MENU_POPUP.in_Rows + INT#02,
// 						Iin_OPTION := INT#00,
// 						Xus_TN_SCREEN := Xus_TN_SCREEN);
//
// 	(* load parameters *)
// 	in_COL := Xus_TN_MENU_POPUP.in_X;
// 	in_ROW := Xus_TN_MENU_POPUP.in_Y;
// 	in_ROWS := Xus_TN_MENU_POPUP.in_Rows;
// 	in_COLS := Xus_TN_MENU_POPUP.in_Cols;
//
// 	(* draw separator lines *)
// 	in_COLS := in_COLS + INT#02; (* extend text by 2 characters *)
//
// 	FOR in_Count := INT#01 TO Xus_TN_MENU_POPUP.in_Menu_E_Count DO;
// 		in_ROW := in_ROW + INT#01;
//
// 		IF ELEMENT_GET(SEP:=BYTE#35,POS:=in_Count - 1,ELEMENT:=Xus_TN_MENU_POPUP.st_Menu_Text) = '-' THEN
//
// 			FB_TN_SC_LINE(	Iin_Y1 := in_ROW,
// 							Iin_X1 := in_COL,
// 							Iin_Y2 := in_ROW,
// 							Iin_X2 := in_COL + in_COLS + INT#01,
// 							Iby_ATTR := Xus_TN_MENU_POPUP.by_Attr_oF,
// 							Iby_BORDER := BYTE#01,
// 							Xus_TN_SCREEN := Xus_TN_SCREEN);
// 		END_IF;
// 	END_FOR;
// END_IF;
//
// IF (Xus_TN_MENU_POPUP.bo_Activ = TRUE) THEN
//
// 	CASE BYTE_TO_INT(Xus_TN_MENU_POPUP.by_Input_Exten_Code) OF
//
// 	65: (* cursor up *)
// 		in_Scroll_Offset := -1;
// 		Xus_TN_MENU_POPUP.bo_Update := TRUE;
//
// 	66: (* cursor down *)
// 		in_Scroll_Offset := 1;
// 		Xus_TN_MENU_POPUP.bo_Update := TRUE;
//
// 	13:  (* Enter *)
// 		Xus_TN_MENU_POPUP.bo_Destroy := TRUE;
//
// 	27:  (* Escape*)
// 		Xus_TN_MENU_POPUP.bo_Destroy := TRUE;
// 		Xus_TN_MENU_POPUP.in_Cur_Item := INT#00;
//
// 	67..68: (* cursor left or right *)
// 		Xus_TN_MENU_POPUP.bo_Destroy := TRUE;
// 		Xus_TN_MENU_POPUP.in_Cur_Item := INT#00;
//
// 	END_CASE;
// END_IF;
//
// (* update POPUP menu *)
// IF (Xus_TN_MENU_POPUP.bo_Activ = TRUE) AND (Xus_TN_MENU_POPUP.bo_Update = TRUE) THEN
//
// 	Xus_TN_MENU_POPUP.bo_Update := FALSE;
//
// 	(* check + find next selectable submenu *)
// 	in_index := Xus_TN_MENU_POPUP.in_Cur_Item;
//
// 	IF (in_index < INT#01) OR (in_index > Xus_TN_MENU_POPUP.in_Menu_E_Count) THEN
// 		in_Scroll_Offset := INT#01;
// 		in_index := Xus_TN_MENU_POPUP.in_Menu_E_Count;
// 	END_IF;
//
// 	(* current index is on a separator -> change *)
// 	IF ELEMENT_GET(SEP:=BYTE#35,POS:=in_index-1,ELEMENT:=Xus_TN_MENU_POPUP.st_Menu_Text) = '-' THEN
// 		in_Scroll_Offset := INT#01;
// 	END_IF;
//
// 	(* Scroll-Offset *)
// 	IF in_Scroll_Offset <> INT#00 THEN
//
// 		FOR in_Count := INT#01 TO Xus_TN_MENU_POPUP.in_Menu_E_Count DO;
//
// 			in_index:=INC2(in_index,in_Scroll_Offset,1,Xus_TN_MENU_POPUP.in_Menu_E_Count);
//
// 			IF ELEMENT_GET(SEP:=BYTE#35,POS:=in_index - 1,ELEMENT:=Xus_TN_MENU_POPUP.st_Menu_Text) <> '-' THEN
// 				EXIT;
// 			END_IF;
//
// 		END_FOR;
// 	END_IF;
//
// 	Xus_TN_MENU_POPUP.in_Cur_Item := in_index;
// 	in_Scroll_Offset := INT#00;
//
// 	(* load parameters *)
// 	in_COL  := Xus_TN_MENU_POPUP.in_X;
// 	in_ROW  := Xus_TN_MENU_POPUP.in_Y;
// 	in_ROWS := Xus_TN_MENU_POPUP.in_Rows;
// 	in_COLS := Xus_TN_MENU_POPUP.in_Cols;
//
// 	(* output SUB-MENU title *)
// 	in_COLS := in_COLS + INT#02; (* extend text by 2 characters *)
//
// 	FOR in_Count := INT#01 TO Xus_TN_MENU_POPUP.in_Menu_E_Count DO;
//
// 		in_ROW := in_ROW + INT#01;
//
// 		(* determine character color *)
// 		IF in_Count = Xus_TN_MENU_POPUP.in_Cur_Item THEN
// 			by_ATTR := Xus_TN_MENU_POPUP.by_Attr_mF;
// 		ELSE
// 			by_ATTR := Xus_TN_MENU_POPUP.by_Attr_oF;
// 		END_IF;
//
// 		FB_TN_SC_WRITE_C.Ist_STRING := ELEMENT_GET(SEP:=BYTE#35,POS:=in_Count - 1,ELEMENT:=Xus_TN_MENU_POPUP.st_Menu_Text);
//
// 		IF FB_TN_SC_WRITE_C.Ist_STRING <> '-' THEN
//
// 			FB_TN_SC_WRITE_C(	Iin_Y := in_ROW,
// 								Iin_X := in_COL + INT#01,
// 								Iby_ATTR := by_ATTR,
// 								Iin_LENGTH := in_COLS,
// 								Iin_OPTION := INT#02, (* Center *)
// 								Xus_TN_SCREEN := Xus_TN_SCREEN);
// 		END_IF;
// 	END_FOR;
// END_IF;
//
// (* remove POPUP menu (destroy) *)
// IF (Xus_TN_MENU_POPUP.bo_Activ = TRUE) AND (Xus_TN_MENU_POPUP.bo_Destroy = TRUE) THEN
//
// 	Xus_TN_MENU_POPUP.bo_Destroy := FALSE;
// 	Xus_TN_MENU_POPUP.bo_Activ := FALSE;
//
// 	(* restore old background from memory *)
// 	FB_TN_SC_AREA_RESTORE(Xus_TN_SCREEN := Xus_TN_SCREEN);
//
// 	Xus_TN_SCREEN.bo_Modal_Dialog := FALSE;
// END_IF;
// END_FUNCTION_BLOCK
